LIN {X 0,Y 556.816,Z 344.275,A -85,B 0,C 180,E1 26754.409,E2 26754.409} C_VEL
LIN {X 0,Y 555.686,Z 542.378,A -85,B 0,C 180,E1 26751.669,E2 26751.669} C_VEL
LIN {X 0,Y 555.397,Z 561.24,A -85,B 0,C 180,E1 26751.213,E2 26751.213} C_VEL
LIN {X 0,Y 554.964,Z 579.491,A -85,B 0,C 180,E1 26750.568,E2 26750.568} C_VEL
LIN {X 0,Y 554.492,Z 596.687,A -85,B 0,C 180,E1 26749.755,E2 26749.755} C_VEL
LIN {X 0,Y 553.933,Z 616.269,A -85,B 0,C 180,E1 26748.582,E2 26748.582} C_VEL
LIN {X 0,Y 553.499,Z 632.409,A -85,B 0,C 180,E1 26747.395,E2 26747.395} C_VEL
LIN {X 0,Y 553.09,Z 647.422,A -85,B 0,C 180,E1 26746.056,E2 26746.056} C_VEL
LIN {X 0,Y 552.732,Z 661.164,A -85,B 0,C 180,E1 26744.582,E2 26744.582} C_VEL
LIN {X 0,Y 552.457,Z 672.902,A -85,B 0,C 180,E1 26743.075,E2 26743.075} C_VEL
LIN {X 0,Y 552.23,Z 683.866,A -85,B 0,C 180,E1 26741.382,E2 26741.382} C_VEL
LIN {X 0,Y 552.076,Z 693.318,A -85,B 0,C 180,E1 26739.591,E2 26739.591} C_VEL
LIN {X 0,Y 551.986,Z 700.982,A -85,B 0,C 180,E1 26737.765,E2 26737.765} C_VEL
LIN {X 0,Y 551.932,Z 707.192,A -85,B 0,C 180,E1 26735.822,E2 26735.822} C_VEL
LIN {X 0,Y 551.92,Z 711.605,A -85,B 0,C 180,E1 26733.843,E2 26733.843} C_VEL
LIN {X 0,Y 551.914,Z 714.178,A -85,B 0,C 180,E1 26731.869,E2 26731.869} C_VEL
LIN {X 0,Y 551.916,Z 714.992,A -85,B 0,C 180,E1 26729.896,E2 26729.896} C_VEL
LIN {X 0,Y 551.917,Z 714.065,A -85,B 0,C 180,E1 26727.924,E2 26727.924} C_VEL
LIN {X 0,Y 551.921,Z 711.376,A -85,B 0,C 180,E1 26725.949,E2 26725.949} C_VEL
LIN {X 0,Y 551.937,Z 706.971,A -85,B 0,C 180,E1 26724.011,E2 26724.011} C_VEL
LIN {X 0,Y 551.988,Z 700.76,A -85,B 0,C 180,E1 26722.088,E2 26722.088} C_VEL
LIN {X 0,Y 552.077,Z 693.245,A -85,B 0,C 180,E1 26720.304,E2 26720.304} C_VEL
LIN {X 0,Y 552.231,Z 683.772,A -85,B 0,C 180,E1 26718.512,E2 26718.512} C_VEL
LIN {X 0,Y 552.458,Z 672.783,A -85,B 0,C 180,E1 26716.819,E2 26716.819} C_VEL
LIN {X 0,Y 552.755,Z 660.265,A -85,B 0,C 180,E1 26715.224,E2 26715.224} C_VEL
LIN {X 0,Y 553.124,Z 646.131,A -85,B 0,C 180,E1 26713.729,E2 26713.729} C_VEL
LIN {X 0,Y 553.539,Z 630.846,A -85,B 0,C 180,E1 26712.389,E2 26712.389} C_VEL
LIN {X 0,Y 553.959,Z 615.253,A -85,B 0,C 180,E1 26711.26,E2 26711.26} C_VEL
LIN {X 0,Y 554.497,Z 596.601,A -85,B 0,C 180,E1 26710.151,E2 26710.151} C_VEL
LIN {X 0,Y 554.987,Z 579.027,A -85,B 0,C 180,E1 26709.323,E2 26709.323} C_VEL
LIN {X 0,Y 555.409,Z 560.565,A -85,B 0,C 180,E1 26708.677,E2 26708.677} C_VEL
LIN {X 0,Y 555.693,Z 541.746,A -85,B 0,C 180,E1 26708.23,E2 26708.23} C_VEL
LIN {X 0,Y 556.819,Z 343.095,A -85,B 0,C 180,E1 26705.485,E2 26705.485} C_VEL
LIN {X 0,Y 555.247,Z 334.788,A -85,B 0,C 180,E1 26705.25,E2 26705.25} C_VEL
LIN {X 0,Y 556.018,Z 305.385,A -85,B 0,C 180,E1 26702.475,E2 26702.475} C_VEL
LIN {X 0,Y 552.345,Z 293.887,A -85,B 0,C 180,E1 26701.069,E2 26701.069} C_VEL
LIN {X 0,Y 552.34,Z 293.681,A -85,B 0,C 180,E1 26697.846,E2 26697.846} C_VEL
LIN {X 0,Y 552.335,Z 293.677,A -85,B 0,C 180,E1 26694.474,E2 26694.474} C_VEL
LIN {X 0,Y 552.308,Z 293.678,A -85,B 0,C 180,E1 26691.119,E2 26691.119} C_VEL
LIN {X 0,Y 552.34,Z 293.682,A -85,B 0,C 180,E1 26687.811,E2 26687.811} C_VEL
LIN {X 0,Y 552.322,Z 293.677,A -85,B 0,C 180,E1 26684.474,E2 26684.474} C_VEL
LIN {X 0,Y 552.301,Z 293.684,A -85,B 0,C 180,E1 26681.084,E2 26681.084} C_VEL
LIN {X 0,Y 552.345,Z 293.682,A -85,B 0,C 180,E1 26677.855,E2 26677.855} C_VEL
LIN {X 0,Y 552.302,Z 293.681,A -85,B 0,C 180,E1 26674.545,E2 26674.545} C_VEL
LIN {X 0,Y 552.297,Z 293.685,A -85,B 0,C 180,E1 26671.099,E2 26671.099} C_VEL
LIN {X 0,Y 552.344,Z 293.681,A -85,B 0,C 180,E1 26667.842,E2 26667.842} C_VEL
LIN {X 0,Y 552.285,Z 293.679,A -85,B 0,C 180,E1 26664.607,E2 26664.607} C_VEL
LIN {X 0,Y 552.314,Z 293.685,A -85,B 0,C 180,E1 26661.338,E2 26661.338} C_VEL
LIN {X 0,Y 552.292,Z 293.682,A -85,B 0,C 180,E1 26658.252,E2 26658.252} C_VEL
LIN {X 0,Y 552.278,Z 293.681,A -85,B 0,C 180,E1 26654.897,E2 26654.897} C_VEL
LIN {X 0,Y 552.337,Z 293.685,A -85,B 0,C 180,E1 26651.676,E2 26651.676} C_VEL
LIN {X 0,Y 552.267,Z 293.68,A -85,B 0,C 180,E1 26648.433,E2 26648.433} C_VEL
LIN {X 0,Y 552.298,Z 293.687,A -85,B 0,C 180,E1 26645.194,E2 26645.194} C_VEL
LIN {X 0,Y 552.276,Z 293.682,A -85,B 0,C 180,E1 26642.075,E2 26642.075} C_VEL
LIN {X 0,Y 552.263,Z 293.686,A -85,B 0,C 180,E1 26638.755,E2 26638.755} C_VEL
LIN {X 0,Y 552.326,Z 293.685,A -85,B 0,C 180,E1 26635.536,E2 26635.536} C_VEL
LIN {X 0,Y 552.265,Z 293.683,A -85,B 0,C 180,E1 26632.406,E2 26632.406} C_VEL
LIN {X 0,Y 552.318,Z 293.686,A -85,B 0,C 180,E1 26629.148,E2 26629.148} C_VEL
LIN {X 0,Y 552.281,Z 293.681,A -85,B 0,C 180,E1 26626.014,E2 26626.014} C_VEL
LIN {X 0,Y 552.279,Z 293.683,A -85,B 0,C 180,E1 26622.566,E2 26622.566} C_VEL
LIN {X 0,Y 552.342,Z 293.686,A -85,B 0,C 180,E1 26619.33,E2 26619.33} C_VEL
LIN {X 0,Y 552.285,Z 293.683,A -85,B 0,C 180,E1 26616.096,E2 26616.096} C_VEL
LIN {X 0,Y 552.309,Z 293.68,A -85,B 0,C 180,E1 26612.741,E2 26612.741} C_VEL
LIN {X 0,Y 552.327,Z 293.686,A -85,B 0,C 180,E1 26609.504,E2 26609.504} C_VEL
LIN {X 0,Y 552.292,Z 293.684,A -85,B 0,C 180,E1 26606.195,E2 26606.195} C_VEL
LIN {X 0,Y 552.345,Z 293.677,A -85,B 0,C 180,E1 26602.93,E2 26602.93} C_VEL
LIN {X 0,Y 552.318,Z 293.684,A -85,B 0,C 180,E1 26599.603,E2 26599.603} C_VEL
LIN {X 0,Y 552.305,Z 293.684,A -85,B 0,C 180,E1 26596.245,E2 26596.245} C_VEL
LIN {X 0,Y 552.341,Z 293.676,A -85,B 0,C 180,E1 26593.002,E2 26593.002} C_VEL
LIN {X 0,Y 552.312,Z 293.674,A -85,B 0,C 180,E1 26589.702,E2 26589.702} C_VEL
LIN {X 0,Y 552.379,Z 293.923,A -85,B 0,C 180,E1 26586.704,E2 26586.704} C_VEL
LIN {X 0,Y 554.146,Z 298.811,A -85,B 0,C 180,E1 26586.242,E2 26586.242} C_VEL
LIN {X 0,Y 559.158,Z 310.667,A -85,B 0,C 180,E1 26585.196,E2 26585.196} C_VEL
LIN {X 0,Y 558.362,Z 353.988,A -85,B 0,C 180,E1 26582.614,E2 26582.614} C_VEL
LIN {X 0,Y 557.656,Z 390.963,A -85,B 0,C 180,E1 26580.436,E2 26580.436} C_VEL
LIN {X 0,Y 558.742,Z 400.337,A -85,B 0,C 180,E1 26580.232,E2 26580.232} C_VEL
LIN {X 0,Y 557.381,Z 635.152,A -85,B 0,C 180,E1 26576.937,E2 26576.937} C_VEL
LIN {X 0,Y 557.116,Z 659.61,A -85,B 0,C 180,E1 26576.529,E2 26576.529} C_VEL
LIN {X 0,Y 556.72,Z 680.633,A -85,B 0,C 180,E1 26575.975,E2 26575.975} C_VEL
LIN {X 0,Y 556.289,Z 700.028,A -85,B 0,C 180,E1 26575.274,E2 26575.274} C_VEL
LIN {X 0,Y 555.753,Z 719.239,A -85,B 0,C 180,E1 26574.386,E2 26574.386} C_VEL
LIN {X 0,Y 555.148,Z 738.316,A -85,B 0,C 180,E1 26573.286,E2 26573.286} C_VEL
LIN {X 0,Y 554.551,Z 756.388,A -85,B 0,C 180,E1 26572.025,E2 26572.025} C_VEL
LIN {X 0,Y 553.976,Z 773.443,A -85,B 0,C 180,E1 26570.606,E2 26570.606} C_VEL
LIN {X 0,Y 553.441,Z 789.448,A -85,B 0,C 180,E1 26569.031,E2 26569.031} C_VEL
LIN {X 0,Y 552.984,Z 804.238,A -85,B 0,C 180,E1 26567.315,E2 26567.315} C_VEL
LIN {X 0,Y 552.622,Z 817.278,A -85,B 0,C 180,E1 26565.531,E2 26565.531} C_VEL
LIN {X 0,Y 552.359,Z 828.534,A -85,B 0,C 180,E1 26563.717,E2 26563.717} C_VEL
LIN {X 0,Y 552.147,Z 838.91,A -85,B 0,C 180,E1 26561.701,E2 26561.701} C_VEL
LIN {X 0,Y 552.024,Z 847.28,A -85,B 0,C 180,E1 26559.697,E2 26559.697} C_VEL
LIN {X 0,Y 551.959,Z 854.202,A -85,B 0,C 180,E1 26557.599,E2 26557.599} C_VEL
LIN {X 0,Y 551.92,Z 859.556,A -85,B 0,C 180,E1 26555.405,E2 26555.405} C_VEL
LIN {X 0,Y 551.909,Z 862.942,A -85,B 0,C 180,E1 26553.323,E2 26553.323} C_VEL
LIN {X 0,Y 551.911,Z 864.759,A -85,B 0,C 180,E1 26551.142,E2 26551.142} C_VEL
LIN {X 0,Y 551.915,Z 864.783,A -85,B 0,C 180,E1 26548.962,E2 26548.962} C_VEL
LIN {X 0,Y 551.914,Z 863.169,A -85,B 0,C 180,E1 26546.885,E2 26546.885} C_VEL
LIN {X 0,Y 551.921,Z 859.76,A -85,B 0,C 180,E1 26544.699,E2 26544.699} C_VEL
LIN {X 0,Y 551.952,Z 854.809,A -85,B 0,C 180,E1 26542.611,E2 26542.611} C_VEL
LIN {X 0,Y 552.022,Z 848.49,A -85,B 0,C 180,E1 26540.618,E2 26540.618} C_VEL
LIN {X 0,Y 552.138,Z 839.875,A -85,B 0,C 180,E1 26538.51,E2 26538.51} C_VEL
LIN {X 0,Y 552.321,Z 830.266,A -85,B 0,C 180,E1 26536.602,E2 26536.602} C_VEL
LIN {X 0,Y 552.585,Z 818.607,A -85,B 0,C 180,E1 26534.67,E2 26534.67} C_VEL
LIN {X 0,Y 552.945,Z 805.602,A -85,B 0,C 180,E1 26532.858,E2 26532.858} C_VEL
LIN {X 0,Y 553.393,Z 790.965,A -85,B 0,C 180,E1 26531.131,E2 26531.131} C_VEL
LIN {X 0,Y 553.892,Z 775.855,A -85,B 0,C 180,E1 26529.611,E2 26529.611} C_VEL
LIN {X 0,Y 554.455,Z 759.284,A -85,B 0,C 180,E1 26528.193,E2 26528.193} C_VEL
LIN {X 0,Y 555.07,Z 740.902,A -85,B 0,C 180,E1 26526.879,E2 26526.879} C_VEL
LIN {X 0,Y 555.652,Z 722.284,A -85,B 0,C 180,E1 26525.779,E2 26525.779} C_VEL
LIN {X 0,Y 556.159,Z 704.004,A -85,B 0,C 180,E1 26524.896,E2 26524.896} C_VEL
LIN {X 0,Y 556.654,Z 683.569,A -85,B 0,C 180,E1 26524.118,E2 26524.118} C_VEL
LIN {X 0,Y 557.081,Z 663.506,A -85,B 0,C 180,E1 26523.556,E2 26523.556} C_VEL
LIN {X 0,Y 557.344,Z 642.37,A -85,B 0,C 180,E1 26523.163,E2 26523.163} C_VEL
LIN {X 0,Y 558.712,Z 404.697,A -85,B 0,C 180,E1 26519.829,E2 26519.829} C_VEL
LIN {X 0,Y 558.481,Z 396.637,A -85,B 0,C 180,E1 26519.698,E2 26519.698} C_VEL
LIN {X 0,Y 557.585,Z 389.593,A -85,B 0,C 180,E1 26519.505,E2 26519.505} C_VEL
LIN {X 0,Y 558.839,Z 332.018,A -85,B 0,C 180,E1 26516.068,E2 26516.068} C_VEL
LIN {X 0,Y 558.964,Z 309.864,A -85,B 0,C 180,E1 26514.743,E2 26514.743} C_VEL
LIN {X 0,Y 552.405,Z 294.092,A -85,B 0,C 180,E1 26513.324,E2 26513.324} C_VEL
LIN {X 0,Y 552.339,Z 293.671,A -85,B 0,C 180,E1 26512.969,E2 26512.969} C_VEL
LIN {X 0,Y 552.316,Z 293.676,A -85,B 0,C 180,E1 26509.653,E2 26509.653} C_VEL
LIN {X 0,Y 552.31,Z 293.676,A -85,B 0,C 180,E1 26506.246,E2 26506.246} C_VEL
LIN {X 0,Y 552.344,Z 293.682,A -85,B 0,C 180,E1 26503.004,E2 26503.004} C_VEL
LIN {X 0,Y 552.302,Z 293.683,A -85,B 0,C 180,E1 26499.702,E2 26499.702} C_VEL
LIN {X 0,Y 552.307,Z 293.672,A -85,B 0,C 180,E1 26496.297,E2 26496.297} C_VEL
LIN {X 0,Y 552.34,Z 293.682,A -85,B 0,C 180,E1 26493.016,E2 26493.016} C_VEL
LIN {X 0,Y 552.29,Z 293.685,A -85,B 0,C 180,E1 26489.739,E2 26489.739} C_VEL
LIN {X 0,Y 552.326,Z 293.687,A -85,B 0,C 180,E1 26486.444,E2 26486.444} C_VEL
LIN {X 0,Y 552.304,Z 293.681,A -85,B 0,C 180,E1 26483.244,E2 26483.244} C_VEL
LIN {X 0,Y 552.284,Z 293.685,A -85,B 0,C 180,E1 26479.898,E2 26479.898} C_VEL
LIN {X 0,Y 552.345,Z 293.684,A -85,B 0,C 180,E1 26476.619,E2 26476.619} C_VEL
LIN {X 0,Y 552.277,Z 293.679,A -85,B 0,C 180,E1 26473.399,E2 26473.399} C_VEL
LIN {X 0,Y 552.284,Z 293.685,A -85,B 0,C 180,E1 26469.992,E2 26469.992} C_VEL
LIN {X 0,Y 552.307,Z 293.682,A -85,B 0,C 180,E1 26466.862,E2 26466.862} C_VEL
LIN {X 0,Y 552.263,Z 293.684,A -85,B 0,C 180,E1 26463.633,E2 26463.633} C_VEL
LIN {X 0,Y 552.332,Z 293.688,A -85,B 0,C 180,E1 26460.415,E2 26460.415} C_VEL
LIN {X 0,Y 552.261,Z 293.683,A -85,B 0,C 180,E1 26457.198,E2 26457.198} C_VEL
LIN {X 0,Y 552.27,Z 293.687,A -85,B 0,C 180,E1 26453.764,E2 26453.764} C_VEL
LIN {X 0,Y 552.286,Z 293.681,A -85,B 0,C 180,E1 26450.833,E2 26450.833} C_VEL
LIN {X 0,Y 552.268,Z 293.686,A -85,B 0,C 180,E1 26447.558,E2 26447.558} C_VEL
LIN {X 0,Y 552.34,Z 293.683,A -85,B 0,C 180,E1 26444.352,E2 26444.352} C_VEL
LIN {X 0,Y 552.276,Z 293.684,A -85,B 0,C 180,E1 26441.091,E2 26441.091} C_VEL
LIN {X 0,Y 552.301,Z 293.685,A -85,B 0,C 180,E1 26437.767,E2 26437.767} C_VEL
LIN {X 0,Y 552.312,Z 293.681,A -85,B 0,C 180,E1 26434.593,E2 26434.593} C_VEL
LIN {X 0,Y 552.299,Z 293.687,A -85,B 0,C 180,E1 26432.738,E2 26432.738} C_VEL
LIN {X 0,Y 551.36,Z 293.809,A -85,B 0,C 180,E1 26431.938,E2 26431.938} C_VEL
LIN {X 0,Y 544.881,Z 294.609,A -85,B 0,C 180,E1 26429.694,E2 26429.694} C_VEL
LIN {X 0,Y 544.346,Z 294.673,A -85,B 0,C 180,E1 26429.109,E2 26429.109} C_VEL
LIN {X 0,Y 544.389,Z 294.67,A -85,B 0,C 180,E1 26425.804,E2 26425.804} C_VEL
LIN {X 0,Y 544.381,Z 294.675,A -85,B 0,C 180,E1 26422.507,E2 26422.507} C_VEL
LIN {X 0,Y 544.357,Z 294.672,A -85,B 0,C 180,E1 26419.164,E2 26419.164} C_VEL
LIN {X 0,Y 544.405,Z 294.667,A -85,B 0,C 180,E1 26415.887,E2 26415.887} C_VEL
LIN {X 0,Y 544.376,Z 294.665,A -85,B 0,C 180,E1 26412.523,E2 26412.523} C_VEL
LIN {X 0,Y 544.368,Z 294.665,A -85,B 0,C 180,E1 26409.184,E2 26409.184} C_VEL
LIN {X 0,Y 544.404,Z 294.669,A -85,B 0,C 180,E1 26405.864,E2 26405.864} C_VEL
LIN {X 0,Y 544.38,Z 294.676,A -85,B 0,C 180,E1 26402.537,E2 26402.537} C_VEL
LIN {X 0,Y 544.416,Z 294.861,A -85,B 0,C 180,E1 26399.297,E2 26399.297} C_VEL
LIN {X 0,Y 548.778,Z 308.855,A -85,B 0,C 180,E1 26397.566,E2 26397.566} C_VEL
LIN {X 0,Y 548.006,Z 335.919,A -85,B 0,C 180,E1 26395.02,E2 26395.02} C_VEL
LIN {X 0,Y 549.744,Z 345.387,A -85,B 0,C 180,E1 26394.785,E2 26394.785} C_VEL
LIN {X 0,Y 548.559,Z 542.987,A -85,B 0,C 180,E1 26392.041,E2 26392.041} C_VEL
LIN {X 0,Y 548.263,Z 561.882,A -85,B 0,C 180,E1 26391.584,E2 26391.584} C_VEL
LIN {X 0,Y 547.817,Z 579.557,A -85,B 0,C 180,E1 26390.96,E2 26390.96} C_VEL
LIN {X 0,Y 547.296,Z 596.827,A -85,B 0,C 180,E1 26390.146,E2 26390.146} C_VEL
LIN {X 0,Y 546.679,Z 613.249,A -85,B 0,C 180,E1 26389.165,E2 26389.165} C_VEL
LIN {X 0,Y 546.031,Z 629.329,A -85,B 0,C 180,E1 26387.971,E2 26387.971} C_VEL
LIN {X 0,Y 545.411,Z 644.251,A -85,B 0,C 180,E1 26386.617,E2 26386.617} C_VEL
LIN {X 0,Y 544.925,Z 659.491,A -85,B 0,C 180,E1 26384.993,E2 26384.993} C_VEL
LIN {X 0,Y 544.571,Z 672.136,A -85,B 0,C 180,E1 26383.376,E2 26383.376} C_VEL
LIN {X 0,Y 544.302,Z 683.234,A -85,B 0,C 180,E1 26381.657,E2 26381.657} C_VEL
LIN {X 0,Y 544.121,Z 692.806,A -85,B 0,C 180,E1 26379.84,E2 26379.84} C_VEL
LIN {X 0,Y 544.003,Z 700.413,A -85,B 0,C 180,E1 26378.029,E2 26378.029} C_VEL
LIN {X 0,Y 543.946,Z 706.59,A -85,B 0,C 180,E1 26376.12,E2 26376.12} C_VEL
LIN {X 0,Y 543.921,Z 710.996,A -85,B 0,C 180,E1 26374.217,E2 26374.217} C_VEL
LIN {X 0,Y 543.913,Z 713.744,A -85,B 0,C 180,E1 26372.318,E2 26372.318} C_VEL
LIN {X 0,Y 543.909,Z 714.928,A -85,B 0,C 180,E1 26370.316,E2 26370.316} C_VEL
LIN {X 0,Y 543.913,Z 714.376,A -85,B 0,C 180,E1 26368.315,E2 26368.315} C_VEL
LIN {X 0,Y 543.911,Z 712.229,A -85,B 0,C 180,E1 26366.417,E2 26366.417} C_VEL
LIN {X 0,Y 543.932,Z 708.459,A -85,B 0,C 180,E1 26364.515,E2 26364.515} C_VEL
LIN {X 0,Y 543.974,Z 702.972,A -85,B 0,C 180,E1 26362.608,E2 26362.608} C_VEL
LIN {X 0,Y 544.075,Z 695.621,A -85,B 0,C 180,E1 26360.694,E2 26360.694} C_VEL
LIN {X 0,Y 544.235,Z 686.506,A -85,B 0,C 180,E1 26358.831,E2 26358.831} C_VEL
LIN {X 0,Y 544.463,Z 676.445,A -85,B 0,C 180,E1 26357.162,E2 26357.162} C_VEL
LIN {X 0,Y 544.769,Z 664.701,A -85,B 0,C 180,E1 26355.546,E2 26355.546} C_VEL
LIN {X 0,Y 545.161,Z 651.496,A -85,B 0,C 180,E1 26354.032,E2 26354.032} C_VEL
LIN {X 0,Y 545.774,Z 635.715,A -85,B 0,C 180,E1 26352.484,E2 26352.484} C_VEL
LIN {X 0,Y 546.393,Z 620.716,A -85,B 0,C 180,E1 26351.268,E2 26351.268} C_VEL
LIN {X 0,Y 547.021,Z 604.25,A -85,B 0,C 180,E1 26350.181,E2 26350.181} C_VEL
LIN {X 0,Y 547.584,Z 587.755,A -85,B 0,C 180,E1 26349.31,E2 26349.31} C_VEL
LIN {X 0,Y 548.078,Z 569.85,A -85,B 0,C 180,E1 26348.584,E2 26348.584} C_VEL
LIN {X 0,Y 548.441,Z 551.518,A -85,B 0,C 180,E1 26348.051,E2 26348.051} C_VEL
LIN {X 0,Y 548.652,Z 532.068,A -85,B 0,C 180,E1 26347.695,E2 26347.695} C_VEL
LIN {X 0,Y 549.626,Z 343.643,A -85,B 0,C 180,E1 26345.094,E2 26345.094} C_VEL
LIN {X 0,Y 547.949,Z 335.49,A -85,B 0,C 180,E1 26344.869,E2 26344.869} C_VEL
LIN {X 0,Y 548.672,Z 308.058,A -85,B 0,C 180,E1 26342.257,E2 26342.257} C_VEL
LIN {X 0,Y 544.419,Z 294.84,A -85,B 0,C 180,E1 26340.606,E2 26340.606} C_VEL
LIN {X 0,Y 544.375,Z 294.675,A -85,B 0,C 180,E1 26337.193,E2 26337.193} C_VEL
LIN {X 0,Y 544.4,Z 294.672,A -85,B 0,C 180,E1 26333.876,E2 26333.876} C_VEL
LIN {X 0,Y 544.393,Z 294.662,A -85,B 0,C 180,E1 26330.48,E2 26330.48} C_VEL
LIN {X 0,Y 544.367,Z 294.663,A -85,B 0,C 180,E1 26327.127,E2 26327.127} C_VEL
LIN {X 0,Y 544.405,Z 294.671,A -85,B 0,C 180,E1 26323.8,E2 26323.8} C_VEL
LIN {X 0,Y 544.381,Z 294.669,A -85,B 0,C 180,E1 26320.418,E2 26320.418} C_VEL
LIN {X 0,Y 544.36,Z 294.674,A -85,B 0,C 180,E1 26317.046,E2 26317.046} C_VEL
LIN {X 0,Y 544.403,Z 294.67,A -85,B 0,C 180,E1 26313.699,E2 26313.699} C_VEL
LIN {X 0,Y 544.361,Z 294.671,A -85,B 0,C 180,E1 26310.461,E2 26310.461} C_VEL
LIN {X 0,Y 544.354,Z 294.675,A -85,B 0,C 180,E1 26307.025,E2 26307.025} C_VEL
LIN {X 0,Y 544.404,Z 294.668,A -85,B 0,C 180,E1 26303.717,E2 26303.717} C_VEL
LIN {X 0,Y 544.345,Z 294.671,A -85,B 0,C 180,E1 26300.488,E2 26300.488} C_VEL
LIN {X 0,Y 544.352,Z 294.676,A -85,B 0,C 180,E1 26297.091,E2 26297.091} C_VEL
LIN {X 0,Y 544.376,Z 294.667,A -85,B 0,C 180,E1 26293.923,E2 26293.923} C_VEL
LIN {X 0,Y 544.33,Z 294.675,A -85,B 0,C 180,E1 26290.676,E2 26290.676} C_VEL
LIN {X 0,Y 544.382,Z 294.675,A -85,B 0,C 180,E1 26287.387,E2 26287.387} C_VEL
LIN {X 0,Y 544.331,Z 294.675,A -85,B 0,C 180,E1 26284.214,E2 26284.214} C_VEL
LIN {X 0,Y 544.328,Z 294.677,A -85,B 0,C 180,E1 26280.842,E2 26280.842} C_VEL
LIN {X 0,Y 544.358,Z 294.674,A -85,B 0,C 180,E1 26277.79,E2 26277.79} C_VEL
LIN {X 0,Y 544.324,Z 294.676,A -85,B 0,C 180,E1 26274.519,E2 26274.519} C_VEL
LIN {X 0,Y 544.394,Z 294.67,A -85,B 0,C 180,E1 26271.338,E2 26271.338} C_VEL
LIN {X 0,Y 544.336,Z 294.676,A -85,B 0,C 180,E1 26268.128,E2 26268.128} C_VEL
LIN {X 0,Y 544.343,Z 294.675,A -85,B 0,C 180,E1 26264.644,E2 26264.644} C_VEL
LIN {X 0,Y 544.4,Z 294.669,A -85,B 0,C 180,E1 26261.382,E2 26261.382} C_VEL
LIN {X 0,Y 544.344,Z 294.675,A -85,B 0,C 180,E1 26258.107,E2 26258.107} C_VEL
LIN {X 0,Y 544.37,Z 294.673,A -85,B 0,C 180,E1 26254.779,E2 26254.779} C_VEL
LIN {X 0,Y 544.38,Z 294.673,A -85,B 0,C 180,E1 26251.595,E2 26251.595} C_VEL
LIN {X 0,Y 544.353,Z 294.672,A -85,B 0,C 180,E1 26248.256,E2 26248.256} C_VEL
LIN {X 0,Y 544.399,Z 294.657,A -85,B 0,C 180,E1 26244.91,E2 26244.91} C_VEL
LIN {X 0,Y 544.377,Z 294.673,A -85,B 0,C 180,E1 26241.625,E2 26241.625} C_VEL
LIN {X 0,Y 544.361,Z 294.657,A -85,B 0,C 180,E1 26238.219,E2 26238.219} C_VEL
LIN {X 0,Y 544.405,Z 294.666,A -85,B 0,C 180,E1 26234.997,E2 26234.997} C_VEL
LIN {X 0,Y 544.379,Z 294.677,A -85,B 0,C 180,E1 26231.623,E2 26231.623} C_VEL
LIN {X 0,Y 544.374,Z 294.678,A -85,B 0,C 180,E1 26228.177,E2 26228.177} C_VEL
LIN {X 0,Y 544.442,Z 294.964,A -85,B 0,C 180,E1 26227.17,E2 26227.17} C_VEL
LIN {X 0,Y 548.919,Z 306.372,A -85,B 0,C 180,E1 26226.115,E2 26226.115} C_VEL
LIN {X 0,Y 552.058,Z 313.827,A -85,B 0,C 180,E1 26225.452,E2 26225.452} C_VEL
LIN {X 0,Y 551.041,Z 367.835,A -85,B 0,C 180,E1 26222.238,E2 26222.238} C_VEL
LIN {X 0,Y 550.595,Z 391.148,A -85,B 0,C 180,E1 26220.865,E2 26220.865} C_VEL
LIN {X 0,Y 551.824,Z 401.323,A -85,B 0,C 180,E1 26220.637,E2 26220.637} C_VEL
LIN {X 0,Y 550.243,Z 636.347,A -85,B 0,C 180,E1 26217.298,E2 26217.298} C_VEL
LIN {X 0,Y 549.945,Z 659.772,A -85,B 0,C 180,E1 26216.898,E2 26216.898} C_VEL
LIN {X 0,Y 549.493,Z 680.847,A -85,B 0,C 180,E1 26216.336,E2 26216.336} C_VEL
LIN {X 0,Y 548.978,Z 700.613,A -85,B 0,C 180,E1 26215.609,E2 26215.609} C_VEL
LIN {X 0,Y 548.378,Z 719.24,A -85,B 0,C 180,E1 26214.736,E2 26214.736} C_VEL
LIN {X 0,Y 547.692,Z 738.326,A -85,B 0,C 180,E1 26213.622,E2 26213.622} C_VEL
LIN {X 0,Y 546.999,Z 756.39,A -85,B 0,C 180,E1 26212.346,E2 26212.346} C_VEL
LIN {X 0,Y 546.323,Z 773.443,A -85,B 0,C 180,E1 26210.908,E2 26210.908} C_VEL
LIN {X 0,Y 545.715,Z 789.202,A -85,B 0,C 180,E1 26209.338,E2 26209.338} C_VEL
LIN {X 0,Y 545.179,Z 803.91,A -85,B 0,C 180,E1 26207.614,E2 26207.614} C_VEL
LIN {X 0,Y 544.775,Z 816.573,A -85,B 0,C 180,E1 26205.87,E2 26205.87} C_VEL
LIN {X 0,Y 544.438,Z 828.535,A -85,B 0,C 180,E1 26203.92,E2 26203.92} C_VEL
LIN {X 0,Y 544.188,Z 838.909,A -85,B 0,C 180,E1 26201.875,E2 26201.875} C_VEL
LIN {X 0,Y 544.043,Z 847.279,A -85,B 0,C 180,E1 26199.841,E2 26199.841} C_VEL
LIN {X 0,Y 543.968,Z 854.202,A -85,B 0,C 180,E1 26197.711,E2 26197.711} C_VEL
LIN {X 0,Y 543.923,Z 859.556,A -85,B 0,C 180,E1 26195.485,E2 26195.485} C_VEL
LIN {X 0,Y 543.909,Z 862.942,A -85,B 0,C 180,E1 26193.372,E2 26193.372} C_VEL
LIN {X 0,Y 543.91,Z 864.759,A -85,B 0,C 180,E1 26191.159,E2 26191.159} C_VEL
LIN {X 0,Y 543.914,Z 864.783,A -85,B 0,C 180,E1 26188.947,E2 26188.947} C_VEL
LIN {X 0,Y 543.913,Z 863.168,A -85,B 0,C 180,E1 26186.839,E2 26186.839} C_VEL
LIN {X 0,Y 543.922,Z 859.761,A -85,B 0,C 180,E1 26184.621,E2 26184.621} C_VEL
LIN {X 0,Y 543.96,Z 854.81,A -85,B 0,C 180,E1 26182.501,E2 26182.501} C_VEL
LIN {X 0,Y 544.038,Z 848.49,A -85,B 0,C 180,E1 26180.479,E2 26180.479} C_VEL
LIN {X 0,Y 544.175,Z 839.876,A -85,B 0,C 180,E1 26178.34,E2 26178.34} C_VEL
LIN {X 0,Y 544.394,Z 830.268,A -85,B 0,C 180,E1 26176.403,E2 26176.403} C_VEL
LIN {X 0,Y 544.705,Z 818.691,A -85,B 0,C 180,E1 26174.455,E2 26174.455} C_VEL
LIN {X 0,Y 545.128,Z 805.601,A -85,B 0,C 180,E1 26172.605,E2 26172.605} C_VEL
LIN {X 0,Y 545.651,Z 790.965,A -85,B 0,C 180,E1 26170.853,E2 26170.853} C_VEL
LIN {X 0,Y 546.252,Z 775.515,A -85,B 0,C 180,E1 26169.282,E2 26169.282} C_VEL
LIN {X 0,Y 546.907,Z 758.842,A -85,B 0,C 180,E1 26167.841,E2 26167.841} C_VEL
LIN {X 0,Y 547.591,Z 740.898,A -85,B 0,C 180,E1 26166.544,E2 26166.544} C_VEL
LIN {X 0,Y 548.224,Z 723.385,A -85,B 0,C 180,E1 26165.492,E2 26165.492} C_VEL
LIN {X 0,Y 548.857,Z 704.001,A -85,B 0,C 180,E1 26164.538,E2 26164.538} C_VEL
LIN {X 0,Y 549.412,Z 683.823,A -85,B 0,C 180,E1 26163.76,E2 26163.76} C_VEL
LIN {X 0,Y 549.903,Z 663.669,A -85,B 0,C 180,E1 26163.187,E2 26163.187} C_VEL
LIN {X 0,Y 550.205,Z 642.495,A -85,B 0,C 180,E1 26162.788,E2 26162.788} C_VEL
LIN {X 0,Y 551.793,Z 405.141,A -85,B 0,C 180,E1 26159.417,E2 26159.417} C_VEL
LIN {X 0,Y 551.569,Z 397.823,A -85,B 0,C 180,E1 26159.295,E2 26159.295} C_VEL
LIN {X 0,Y 550.502,Z 389.593,A -85,B 0,C 180,E1 26159.07,E2 26159.07} C_VEL
LIN {X 0,Y 551.484,Z 344.188,A -85,B 0,C 180,E1 26156.367,E2 26156.367} C_VEL
LIN {X 0,Y 551.986,Z 313.279,A -85,B 0,C 180,E1 26154.51,E2 26154.51} C_VEL
LIN {X 0,Y 544.464,Z 295.085,A -85,B 0,C 180,E1 26152.844,E2 26152.844} C_VEL
LIN {X 0,Y 544.387,Z 294.664,A -85,B 0,C 180,E1 26152.508,E2 26152.508} C_VEL
LIN {X 0,Y 544.405,Z 294.663,A -85,B 0,C 180,E1 26149.17,E2 26149.17} C_VEL
LIN {X 0,Y 544.365,Z 294.666,A -85,B 0,C 180,E1 26145.885,E2 26145.885} C_VEL
LIN {X 0,Y 544.388,Z 294.66,A -85,B 0,C 180,E1 26142.523,E2 26142.523} C_VEL
LIN {X 0,Y 544.401,Z 294.67,A -85,B 0,C 180,E1 26139.183,E2 26139.183} C_VEL
LIN {X 0,Y 544.354,Z 294.66,A -85,B 0,C 180,E1 26135.869,E2 26135.869} C_VEL
LIN {X 0,Y 544.393,Z 294.676,A -85,B 0,C 180,E1 26132.542,E2 26132.542} C_VEL
LIN {X 0,Y 544.376,Z 294.672,A -85,B 0,C 180,E1 26129.246,E2 26129.246} C_VEL
LIN {X 0,Y 544.349,Z 294.675,A -85,B 0,C 180,E1 26125.922,E2 26125.922} C_VEL
LIN {X 0,Y 544.409,Z 294.668,A -85,B 0,C 180,E1 26122.686,E2 26122.686} C_VEL
LIN {X 0,Y 544.348,Z 294.672,A -85,B 0,C 180,E1 26119.418,E2 26119.418} C_VEL
LIN {X 0,Y 544.349,Z 294.676,A -85,B 0,C 180,E1 26115.993,E2 26115.993} C_VEL
LIN {X 0,Y 544.397,Z 294.666,A -85,B 0,C 180,E1 26112.732,E2 26112.732} C_VEL
LIN {X 0,Y 544.333,Z 294.673,A -85,B 0,C 180,E1 26109.474,E2 26109.474} C_VEL
LIN {X 0,Y 544.366,Z 294.677,A -85,B 0,C 180,E1 26106.221,E2 26106.221} C_VEL
LIN {X 0,Y 544.342,Z 294.672,A -85,B 0,C 180,E1 26103.053,E2 26103.053} C_VEL
LIN {X 0,Y 544.324,Z 294.677,A -85,B 0,C 180,E1 26099.684,E2 26099.684} C_VEL
LIN {X 0,Y 544.383,Z 294.669,A -85,B 0,C 180,E1 26096.525,E2 26096.525} C_VEL
LIN {X 0,Y 544.321,Z 294.676,A -85,B 0,C 180,E1 26093.354,E2 26093.354} C_VEL
LIN {X 0,Y 544.376,Z 294.675,A -85,B 0,C 180,E1 26090.165,E2 26090.165} C_VEL
LIN {X 0,Y 544.335,Z 294.675,A -85,B 0,C 180,E1 26087.05,E2 26087.05} C_VEL
LIN {X 0,Y 544.338,Z 294.675,A -85,B 0,C 180,E1 26083.568,E2 26083.568} C_VEL
LIN {X 0,Y 544.397,Z 294.669,A -85,B 0,C 180,E1 26080.36,E2 26080.36} C_VEL
LIN {X 0,Y 544.34,Z 294.675,A -85,B 0,C 180,E1 26077.082,E2 26077.082} C_VEL
LIN {X 0,Y 544.361,Z 294.673,A -85,B 0,C 180,E1 26073.677,E2 26073.677} C_VEL
LIN {X 0,Y 544.38,Z 294.672,A -85,B 0,C 180,E1 26070.512,E2 26070.512} C_VEL
LIN {X 0,Y 544.346,Z 294.673,A -85,B 0,C 180,E1 26069.109,E2 26069.109} C_VEL
LIN {X 0,Y 543.375,Z 294.804,A -85,B 0,C 180,E1 26068.298,E2 26068.298} C_VEL
LIN {X 0,Y 536.878,Z 295.607,A -85,B 0,C 180,E1 26065.962,E2 26065.962} C_VEL
LIN {X 0,Y 536.42,Z 295.66,A -85,B 0,C 180,E1 26065.427,E2 26065.427} C_VEL
LIN {X 0,Y 536.466,Z 295.659,A -85,B 0,C 180,E1 26062.179,E2 26062.179} C_VEL
LIN {X 0,Y 536.421,Z 295.663,A -85,B 0,C 180,E1 26058.852,E2 26058.852} C_VEL
LIN {X 0,Y 536.433,Z 295.656,A -85,B 0,C 180,E1 26055.397,E2 26055.397} C_VEL
LIN {X 0,Y 536.464,Z 295.657,A -85,B 0,C 180,E1 26052.116,E2 26052.116} C_VEL
LIN {X 0,Y 536.426,Z 295.652,A -85,B 0,C 180,E1 26048.775,E2 26048.775} C_VEL
LIN {X 0,Y 536.442,Z 295.657,A -85,B 0,C 180,E1 26045.295,E2 26045.295} C_VEL
LIN {X 0,Y 536.463,Z 295.656,A -85,B 0,C 180,E1 26041.958,E2 26041.958} C_VEL
LIN {X 0,Y 536.499,Z 295.915,A -85,B 0,C 180,E1 26039.745,E2 26039.745} C_VEL
LIN {X 0,Y 541.485,Z 311.262,A -85,B 0,C 180,E1 26037.812,E2 26037.812} C_VEL
LIN {X 0,Y 540.72,Z 336.313,A -85,B 0,C 180,E1 26035.435,E2 26035.435} C_VEL
LIN {X 0,Y 542.697,Z 346.672,A -85,B 0,C 180,E1 26035.169,E2 26035.169} C_VEL
LIN {X 0,Y 541.466,Z 544.211,A -85,B 0,C 180,E1 26032.415,E2 26032.415} C_VEL
LIN {X 0,Y 541.155,Z 563.162,A -85,B 0,C 180,E1 26031.949,E2 26031.949} C_VEL
LIN {X 0,Y 540.667,Z 580.996,A -85,B 0,C 180,E1 26031.308,E2 26031.308} C_VEL
LIN {X 0,Y 540.083,Z 598.216,A -85,B 0,C 180,E1 26030.48,E2 26030.48} C_VEL
LIN {X 0,Y 539.356,Z 615.276,A -85,B 0,C 180,E1 26029.436,E2 26029.436} C_VEL
LIN {X 0,Y 538.667,Z 630.549,A -85,B 0,C 180,E1 26028.281,E2 26028.281} C_VEL
LIN {X 0,Y 537.958,Z 645.447,A -85,B 0,C 180,E1 26026.91,E2 26026.91} C_VEL
LIN {X 0,Y 537.315,Z 658.759,A -85,B 0,C 180,E1 26025.432,E2 26025.432} C_VEL
LIN {X 0,Y 536.769,Z 671.005,A -85,B 0,C 180,E1 26023.794,E2 26023.794} C_VEL
LIN {X 0,Y 536.337,Z 684.507,A -85,B 0,C 180,E1 26021.615,E2 26021.615} C_VEL
LIN {X 0,Y 536.133,Z 693.838,A -85,B 0,C 180,E1 26019.771,E2 26019.771} C_VEL
LIN {X 0,Y 536.006,Z 701.614,A -85,B 0,C 180,E1 26017.826,E2 26017.826} C_VEL
LIN {X 0,Y 535.94,Z 707.481,A -85,B 0,C 180,E1 26015.889,E2 26015.889} C_VEL
LIN {X 0,Y 535.92,Z 711.772,A -85,B 0,C 180,E1 26013.851,E2 26013.851} C_VEL
LIN {X 0,Y 535.913,Z 714.248,A -85,B 0,C 180,E1 26011.818,E2 26011.818} C_VEL
LIN {X 0,Y 535.913,Z 714.969,A -85,B 0,C 180,E1 26009.786,E2 26009.786} C_VEL
LIN {X 0,Y 535.916,Z 713.954,A -85,B 0,C 180,E1 26007.755,E2 26007.755} C_VEL
LIN {X 0,Y 535.922,Z 711.375,A -85,B 0,C 180,E1 26005.828,E2 26005.828} C_VEL
LIN {X 0,Y 535.947,Z 707.148,A -85,B 0,C 180,E1 26003.896,E2 26003.896} C_VEL
LIN {X 0,Y 536.013,Z 701.161,A -85,B 0,C 180,E1 26001.958,E2 26001.958} C_VEL
LIN {X 0,Y 536.136,Z 693.754,A -85,B 0,C 180,E1 26000.121,E2 26000.121} C_VEL
LIN {X 0,Y 536.341,Z 684.398,A -85,B 0,C 180,E1 25998.276,E2 25998.276} C_VEL
LIN {X 0,Y 536.794,Z 670.46,A -85,B 0,C 180,E1 25996.035,E2 25996.035} C_VEL
LIN {X 0,Y 537.325,Z 658.594,A -85,B 0,C 180,E1 25994.458,E2 25994.458} C_VEL
LIN {X 0,Y 537.971,Z 645.245,A -85,B 0,C 180,E1 25992.979,E2 25992.979} C_VEL
LIN {X 0,Y 538.681,Z 630.3,A -85,B 0,C 180,E1 25991.607,E2 25991.607} C_VEL
LIN {X 0,Y 539.414,Z 614.175,A -85,B 0,C 180,E1 25990.398,E2 25990.398} C_VEL
LIN {X 0,Y 540.101,Z 597.813,A -85,B 0,C 180,E1 25989.407,E2 25989.407} C_VEL
LIN {X 0,Y 540.692,Z 580.44,A -85,B 0,C 180,E1 25988.579,E2 25988.579} C_VEL
LIN {X 0,Y 541.172,Z 562.076,A -85,B 0,C 180,E1 25987.93,E2 25987.93} C_VEL
LIN {X 0,Y 541.473,Z 543.525,A -85,B 0,C 180,E1 25987.484,E2 25987.484} C_VEL
LIN {X 0,Y 542.586,Z 364.02,A -85,B 0,C 180,E1 25984.978,E2 25984.978} C_VEL
LIN {X 0,Y 542.483,Z 344.395,A -85,B 0,C 180,E1 25984.696,E2 25984.696} C_VEL
LIN {X 0,Y 540.658,Z 335.774,A -85,B 0,C 180,E1 25984.445,E2 25984.445} C_VEL
LIN {X 0,Y 541.472,Z 311.202,A -85,B 0,C 180,E1 25982.09,E2 25982.09} C_VEL
LIN {X 0,Y 536.494,Z 295.899,A -85,B 0,C 180,E1 25980.159,E2 25980.159} C_VEL
LIN {X 0,Y 536.439,Z 295.662,A -85,B 0,C 180,E1 25976.9,E2 25976.9} C_VEL
LIN {X 0,Y 536.442,Z 295.663,A -85,B 0,C 180,E1 25973.386,E2 25973.386} C_VEL
LIN {X 0,Y 536.462,Z 295.654,A -85,B 0,C 180,E1 25969.985,E2 25969.985} C_VEL
LIN {X 0,Y 536.436,Z 295.648,A -85,B 0,C 180,E1 25966.629,E2 25966.629} C_VEL
LIN {X 0,Y 536.428,Z 295.664,A -85,B 0,C 180,E1 25963.162,E2 25963.162} C_VEL
LIN {X 0,Y 536.467,Z 295.661,A -85,B 0,C 180,E1 25959.838,E2 25959.838} C_VEL
LIN {X 0,Y 536.431,Z 295.66,A -85,B 0,C 180,E1 25956.484,E2 25956.484} C_VEL
LIN {X 0,Y 536.42,Z 295.663,A -85,B 0,C 180,E1 25953.103,E2 25953.103} C_VEL
LIN {X 0,Y 536.469,Z 295.658,A -85,B 0,C 180,E1 25949.844,E2 25949.844} C_VEL
LIN {X 0,Y 536.413,Z 295.662,A -85,B 0,C 180,E1 25946.533,E2 25946.533} C_VEL
LIN {X 0,Y 536.414,Z 295.664,A -85,B 0,C 180,E1 25943.044,E2 25943.044} C_VEL
LIN {X 0,Y 536.466,Z 295.656,A -85,B 0,C 180,E1 25939.749,E2 25939.749} C_VEL
LIN {X 0,Y 536.401,Z 295.663,A -85,B 0,C 180,E1 25936.459,E2 25936.459} C_VEL
LIN {X 0,Y 536.407,Z 295.664,A -85,B 0,C 180,E1 25933.035,E2 25933.035} C_VEL
LIN {X 0,Y 536.433,Z 295.663,A -85,B 0,C 180,E1 25929.874,E2 25929.874} C_VEL
LIN {X 0,Y 536.387,Z 295.665,A -85,B 0,C 180,E1 25926.637,E2 25926.637} C_VEL
LIN {X 0,Y 536.443,Z 295.657,A -85,B 0,C 180,E1 25923.42,E2 25923.42} C_VEL
LIN {X 0,Y 536.385,Z 295.666,A -85,B 0,C 180,E1 25920.214,E2 25920.214} C_VEL
LIN {X 0,Y 536.39,Z 295.661,A -85,B 0,C 180,E1 25916.794,E2 25916.794} C_VEL
LIN {X 0,Y 536.446,Z 295.665,A -85,B 0,C 180,E1 25913.579,E2 25913.579} C_VEL
LIN {X 0,Y 536.39,Z 295.663,A -85,B 0,C 180,E1 25910.342,E2 25910.342} C_VEL
LIN {X 0,Y 536.435,Z 295.655,A -85,B 0,C 180,E1 25907.076,E2 25907.076} C_VEL
LIN {X 0,Y 536.414,Z 295.665,A -85,B 0,C 180,E1 25903.875,E2 25903.875} C_VEL
LIN {X 0,Y 536.405,Z 295.662,A -85,B 0,C 180,E1 25900.509,E2 25900.509} C_VEL
LIN {X 0,Y 536.467,Z 295.656,A -85,B 0,C 180,E1 25897.191,E2 25897.191} C_VEL
LIN {X 0,Y 536.417,Z 295.664,A -85,B 0,C 180,E1 25893.903,E2 25893.903} C_VEL
LIN {X 0,Y 536.42,Z 295.662,A -85,B 0,C 180,E1 25890.509,E2 25890.509} C_VEL
LIN {X 0,Y 536.468,Z 295.662,A -85,B 0,C 180,E1 25887.197,E2 25887.197} C_VEL
LIN {X 0,Y 536.419,Z 295.646,A -85,B 0,C 180,E1 25883.914,E2 25883.914} C_VEL
LIN {X 0,Y 536.434,Z 295.66,A -85,B 0,C 180,E1 25880.501,E2 25880.501} C_VEL
LIN {X 0,Y 536.463,Z 295.652,A -85,B 0,C 180,E1 25877.134,E2 25877.134} C_VEL
LIN {X 0,Y 536.432,Z 295.65,A -85,B 0,C 180,E1 25873.748,E2 25873.748} C_VEL
LIN {X 0,Y 536.436,Z 295.65,A -85,B 0,C 180,E1 25870.297,E2 25870.297} C_VEL
LIN {X 0,Y 536.468,Z 295.89,A -85,B 0,C 180,E1 25867.684,E2 25867.684} C_VEL
LIN {X 0,Y 537.386,Z 298.529,A -85,B 0,C 180,E1 25867.395,E2 25867.395} C_VEL
LIN {X 0,Y 544.954,Z 316.732,A -85,B 0,C 180,E1 25865.725,E2 25865.725} C_VEL
LIN {X 0,Y 543.784,Z 370.83,A -85,B 0,C 180,E1 25862.472,E2 25862.472} C_VEL
LIN {X 0,Y 543.515,Z 391.139,A -85,B 0,C 180,E1 25861.306,E2 25861.306} C_VEL
LIN {X 0,Y 544.931,Z 402.537,A -85,B 0,C 180,E1 25861.049,E2 25861.049} C_VEL
LIN {X 0,Y 543.124,Z 637.969,A -85,B 0,C 180,E1 25857.663,E2 25857.663} C_VEL
LIN {X 0,Y 542.789,Z 660.42,A -85,B 0,C 180,E1 25857.267,E2 25857.267} C_VEL
LIN {X 0,Y 542.279,Z 681.388,A -85,B 0,C 180,E1 25856.695,E2 25856.695} C_VEL
LIN {X 0,Y 541.676,Z 701.436,A -85,B 0,C 180,E1 25855.942,E2 25855.942} C_VEL
LIN {X 0,Y 540.985,Z 720.276,A -85,B 0,C 180,E1 25855.039,E2 25855.039} C_VEL
LIN {X 0,Y 540.22,Z 739.219,A -85,B 0,C 180,E1 25853.911,E2 25853.911} C_VEL
LIN {X 0,Y 539.435,Z 757.064,A -85,B 0,C 180,E1 25852.623,E2 25852.623} C_VEL
LIN {X 0,Y 538.666,Z 774.049,A -85,B 0,C 180,E1 25851.163,E2 25851.163} C_VEL
LIN {X 0,Y 537.963,Z 789.953,A -85,B 0,C 180,E1 25849.544,E2 25849.544} C_VEL
LIN {X 0,Y 537.346,Z 804.756,A -85,B 0,C 180,E1 25847.767,E2 25847.767} C_VEL
LIN {X 0,Y 536.86,Z 817.987,A -85,B 0,C 180,E1 25845.889,E2 25845.889} C_VEL
LIN {X 0,Y 536.505,Z 829.114,A -85,B 0,C 180,E1 25844.02,E2 25844.02} C_VEL
LIN {X 0,Y 536.225,Z 839.412,A -85,B 0,C 180,E1 25841.945,E2 25841.945} C_VEL
LIN {X 0,Y 536.056,Z 848.088,A -85,B 0,C 180,E1 25839.772,E2 25839.772} C_VEL
LIN {X 0,Y 535.974,Z 854.505,A -85,B 0,C 180,E1 25837.719,E2 25837.719} C_VEL
LIN {X 0,Y 535.928,Z 859.555,A -85,B 0,C 180,E1 25835.567,E2 25835.567} C_VEL
LIN {X 0,Y 535.91,Z 862.941,A -85,B 0,C 180,E1 25833.423,E2 25833.423} C_VEL
LIN {X 0,Y 535.909,Z 864.759,A -85,B 0,C 180,E1 25831.176,E2 25831.176} C_VEL
LIN {X 0,Y 535.915,Z 864.805,A -85,B 0,C 180,E1 25829.038,E2 25829.038} C_VEL
LIN {X 0,Y 535.914,Z 863.281,A -85,B 0,C 180,E1 25826.899,E2 25826.899} C_VEL
LIN {X 0,Y 535.924,Z 859.966,A -85,B 0,C 180,E1 25824.648,E2 25824.648} C_VEL
LIN {X 0,Y 535.965,Z 855.113,A -85,B 0,C 180,E1 25822.497,E2 25822.497} C_VEL
LIN {X 0,Y 536.055,Z 848.49,A -85,B 0,C 180,E1 25820.336,E2 25820.336} C_VEL
LIN {X 0,Y 536.214,Z 839.877,A -85,B 0,C 180,E1 25818.164,E2 25818.164} C_VEL
LIN {X 0,Y 536.475,Z 830.125,A -85,B 0,C 180,E1 25816.171,E2 25816.171} C_VEL
LIN {X 0,Y 536.835,Z 818.69,A -85,B 0,C 180,E1 25814.222,E2 25814.222} C_VEL
LIN {X 0,Y 537.324,Z 805.371,A -85,B 0,C 180,E1 25812.313,E2 25812.313} C_VEL
LIN {X 0,Y 537.923,Z 790.965,A -85,B 0,C 180,E1 25810.567,E2 25810.567} C_VEL
LIN {X 0,Y 538.596,Z 775.859,A -85,B 0,C 180,E1 25809.006,E2 25809.006} C_VEL
LIN {X 0,Y 539.375,Z 758.573,A -85,B 0,C 180,E1 25807.494,E2 25807.494} C_VEL
LIN {X 0,Y 540.137,Z 740.895,A -85,B 0,C 180,E1 25806.201,E2 25806.201} C_VEL
LIN {X 0,Y 540.87,Z 722.982,A -85,B 0,C 180,E1 25805.114,E2 25805.114} C_VEL
LIN {X 0,Y 541.577,Z 703.998,A -85,B 0,C 180,E1 25804.171,E2 25804.171} C_VEL
LIN {X 0,Y 542.2,Z 683.938,A -85,B 0,C 180,E1 25803.387,E2 25803.387} C_VEL
LIN {X 0,Y 542.749,Z 663.832,A -85,B 0,C 180,E1 25802.808,E2 25802.808} C_VEL
LIN {X 0,Y 543.092,Z 642.495,A -85,B 0,C 180,E1 25802.402,E2 25802.402} C_VEL
LIN {X 0,Y 544.906,Z 405.395,A -85,B 0,C 180,E1 25798.992,E2 25798.992} C_VEL
LIN {X 0,Y 544.666,Z 398.89,A -85,B 0,C 180,E1 25798.879,E2 25798.879} C_VEL
LIN {X 0,Y 543.416,Z 389.969,A -85,B 0,C 180,E1 25798.652,E2 25798.652} C_VEL
LIN {X 0,Y 544.565,Z 334.264,A -85,B 0,C 180,E1 25795.341,E2 25795.341} C_VEL
LIN {X 0,Y 544.752,Z 316.051,A -85,B 0,C 180,E1 25794.219,E2 25794.219} C_VEL
LIN {X 0,Y 536.504,Z 296.088,A -85,B 0,C 180,E1 25792.353,E2 25792.353} C_VEL
LIN {X 0,Y 536.431,Z 295.662,A -85,B 0,C 180,E1 25792.039,E2 25792.039} C_VEL
LIN {X 0,Y 536.464,Z 295.66,A -85,B 0,C 180,E1 25788.686,E2 25788.686} C_VEL
LIN {X 0,Y 536.462,Z 295.652,A -85,B 0,C 180,E1 25785.211,E2 25785.211} C_VEL
LIN {X 0,Y 536.422,Z 295.643,A -85,B 0,C 180,E1 25781.858,E2 25781.858} C_VEL
LIN {X 0,Y 536.448,Z 295.662,A -85,B 0,C 180,E1 25778.483,E2 25778.483} C_VEL
LIN {X 0,Y 536.458,Z 295.644,A -85,B 0,C 180,E1 25775.096,E2 25775.096} C_VEL
LIN {X 0,Y 536.415,Z 295.661,A -85,B 0,C 180,E1 25771.795,E2 25771.795} C_VEL
LIN {X 0,Y 536.455,Z 295.662,A -85,B 0,C 180,E1 25768.499,E2 25768.499} C_VEL
LIN {X 0,Y 536.439,Z 295.662,A -85,B 0,C 180,E1 25765.148,E2 25765.148} C_VEL
LIN {X 0,Y 536.407,Z 295.664,A -85,B 0,C 180,E1 25761.838,E2 25761.838} C_VEL
LIN {X 0,Y 536.461,Z 295.657,A -85,B 0,C 180,E1 25758.585,E2 25758.585} C_VEL
LIN {X 0,Y 536.406,Z 295.663,A -85,B 0,C 180,E1 25755.348,E2 25755.348} C_VEL
LIN {X 0,Y 536.4,Z 295.665,A -85,B 0,C 180,E1 25751.88,E2 25751.88} C_VEL
LIN {X 0,Y 536.459,Z 295.657,A -85,B 0,C 180,E1 25748.575,E2 25748.575} C_VEL
LIN {X 0,Y 536.391,Z 295.665,A -85,B 0,C 180,E1 25745.348,E2 25745.348} C_VEL
LIN {X 0,Y 536.4,Z 295.663,A -85,B 0,C 180,E1 25741.923,E2 25741.923} C_VEL
LIN {X 0,Y 536.415,Z 295.666,A -85,B 0,C 180,E1 25738.825,E2 25738.825} C_VEL
LIN {X 0,Y 536.38,Z 295.665,A -85,B 0,C 180,E1 25735.509,E2 25735.509} C_VEL
LIN {X 0,Y 536.449,Z 295.656,A -85,B 0,C 180,E1 25732.288,E2 25732.288} C_VEL
LIN {X 0,Y 536.396,Z 295.665,A -85,B 0,C 180,E1 25729.039,E2 25729.039} C_VEL
LIN {X 0,Y 536.399,Z 295.657,A -85,B 0,C 180,E1 25725.646,E2 25725.646} C_VEL
LIN {X 0,Y 536.453,Z 295.665,A -85,B 0,C 180,E1 25722.426,E2 25722.426} C_VEL
LIN {X 0,Y 536.399,Z 295.661,A -85,B 0,C 180,E1 25719.143,E2 25719.143} C_VEL
LIN {X 0,Y 536.427,Z 295.655,A -85,B 0,C 180,E1 25715.791,E2 25715.791} C_VEL
LIN {X 0,Y 536.442,Z 295.665,A -85,B 0,C 180,E1 25712.521,E2 25712.521} C_VEL
LIN {X 0,Y 536.408,Z 295.662,A -85,B 0,C 180,E1 25709.235,E2 25709.235} C_VEL
LIN {X 0,Y 536.462,Z 295.658,A -85,B 0,C 180,E1 25706.003,E2 25706.003} C_VEL
LIN {X 0,Y 536.42,Z 295.66,A -85,B 0,C 180,E1 25705.427,E2 25705.427} C_VEL
LIN {X 0,Y 535.423,Z 295.79,A -85,B 0,C 180,E1 25704.605,E2 25704.605} C_VEL
LIN {X 0,Y 528.977,Z 296.593,A -85,B 0,C 180,E1 25702.234,E2 25702.234} C_VEL
LIN {X 0,Y 528.507,Z 296.648,A -85,B 0,C 180,E1 25701.691,E2 25701.691} C_VEL
LIN {X 0,Y 528.517,Z 296.649,A -85,B 0,C 180,E1 25698.353,E2 25698.353} C_VEL
LIN {X 0,Y 528.483,Z 296.646,A -85,B 0,C 180,E1 25694.961,E2 25694.961} C_VEL
LIN {X 0,Y 528.518,Z 296.65,A -85,B 0,C 180,E1 25691.606,E2 25691.606} C_VEL
LIN {X 0,Y 528.523,Z 296.635,A -85,B 0,C 180,E1 25688.214,E2 25688.214} C_VEL
LIN {X 0,Y 528.49,Z 296.642,A -85,B 0,C 180,E1 25684.805,E2 25684.805} C_VEL
LIN {X 0,Y 528.511,Z 296.637,A -85,B 0,C 180,E1 25681.348,E2 25681.348} C_VEL
LIN {X 0,Y 528.551,Z 296.858,A -85,B 0,C 180,E1 25680.242,E2 25680.242} C_VEL
LIN {X 0,Y 534.193,Z 314.111,A -85,B 0,C 180,E1 25678.021,E2 25678.021} C_VEL
LIN {X 0,Y 533.42,Z 336.395,A -85,B 0,C 180,E1 25675.877,E2 25675.877} C_VEL
LIN {X 0,Y 535.67,Z 347.817,A -85,B 0,C 180,E1 25675.564,E2 25675.564} C_VEL
LIN {X 0,Y 534.4,Z 545.275,A -85,B 0,C 180,E1 25672.802,E2 25672.802} C_VEL
LIN {X 0,Y 534.083,Z 564.213,A -85,B 0,C 180,E1 25672.332,E2 25672.332} C_VEL
LIN {X 0,Y 533.546,Z 582.504,A -85,B 0,C 180,E1 25671.664,E2 25671.664} C_VEL
LIN {X 0,Y 532.91,Z 599.652,A -85,B 0,C 180,E1 25670.826,E2 25670.826} C_VEL
LIN {X 0,Y 532.155,Z 615.873,A -85,B 0,C 180,E1 25669.824,E2 25669.824} C_VEL
LIN {X 0,Y 531.335,Z 631.837,A -85,B 0,C 180,E1 25668.6,E2 25668.6} C_VEL
LIN {X 0,Y 530.562,Z 646.088,A -85,B 0,C 180,E1 25667.271,E2 25667.271} C_VEL
LIN {X 0,Y 529.803,Z 659.701,A -85,B 0,C 180,E1 25665.742,E2 25665.742} C_VEL
LIN {X 0,Y 529.169,Z 671.804,A -85,B 0,C 180,E1 25664.107,E2 25664.107} C_VEL
LIN {X 0,Y 528.672,Z 682.608,A -85,B 0,C 180,E1 25662.34,E2 25662.34} C_VEL
LIN {X 0,Y 528.292,Z 691.95,A -85,B 0,C 180,E1 25660.468,E2 25660.468} C_VEL
LIN {X 0,Y 528.065,Z 699.796,A -85,B 0,C 180,E1 25658.493,E2 25658.493} C_VEL
LIN {X 0,Y 527.955,Z 706.594,A -85,B 0,C 180,E1 25656.306,E2 25656.306} C_VEL
LIN {X 0,Y 527.924,Z 710.997,A -85,B 0,C 180,E1 25654.345,E2 25654.345} C_VEL
LIN {X 0,Y 527.911,Z 713.744,A -85,B 0,C 180,E1 25652.388,E2 25652.388} C_VEL
LIN {X 0,Y 527.909,Z 714.927,A -85,B 0,C 180,E1 25650.326,E2 25650.326} C_VEL
LIN {X 0,Y 527.913,Z 714.374,A -85,B 0,C 180,E1 25648.264,E2 25648.264} C_VEL
LIN {X 0,Y 527.914,Z 712.226,A -85,B 0,C 180,E1 25646.308,E2 25646.308} C_VEL
LIN {X 0,Y 527.937,Z 708.455,A -85,B 0,C 180,E1 25644.348,E2 25644.348} C_VEL
LIN {X 0,Y 528.008,Z 702.639,A -85,B 0,C 180,E1 25642.274,E2 25642.274} C_VEL
LIN {X 0,Y 528.172,Z 695.607,A -85,B 0,C 180,E1 25640.301,E2 25640.301} C_VEL
LIN {X 0,Y 528.475,Z 687.161,A -85,B 0,C 180,E1 25638.431,E2 25638.431} C_VEL
LIN {X 0,Y 528.915,Z 677.344,A -85,B 0,C 180,E1 25636.666,E2 25636.666} C_VEL
LIN {X 0,Y 529.452,Z 666.189,A -85,B 0,C 180,E1 25635.006,E2 25635.006} C_VEL
LIN {X 0,Y 530.138,Z 653.641,A -85,B 0,C 180,E1 25633.454,E2 25633.454} C_VEL
LIN {X 0,Y 530.911,Z 639.573,A -85,B 0,C 180,E1 25632.002,E2 25632.002} C_VEL
LIN {X 0,Y 531.708,Z 624.712,A -85,B 0,C 180,E1 25630.734,E2 25630.734} C_VEL
LIN {X 0,Y 532.497,Z 608.695,A -85,B 0,C 180,E1 25629.617,E2 25629.617} C_VEL
LIN {X 0,Y 533.226,Z 591.689,A -85,B 0,C 180,E1 25628.669,E2 25628.669} C_VEL
LIN {X 0,Y 533.817,Z 574.117,A -85,B 0,C 180,E1 25627.914,E2 25627.914} C_VEL
LIN {X 0,Y 534.248,Z 555.617,A -85,B 0,C 180,E1 25627.338,E2 25627.338} C_VEL
LIN {X 0,Y 534.478,Z 536.527,A -85,B 0,C 180,E1 25626.962,E2 25626.962} C_VEL
LIN {X 0,Y 535.554,Z 346.222,A -85,B 0,C 180,E1 25624.316,E2 25624.316} C_VEL
LIN {X 0,Y 533.396,Z 336.077,A -85,B 0,C 180,E1 25624.011,E2 25624.011} C_VEL
LIN {X 0,Y 534.104,Z 313.814,A -85,B 0,C 180,E1 25621.852,E2 25621.852} C_VEL
LIN {X 0,Y 528.55,Z 296.845,A -85,B 0,C 180,E1 25619.664,E2 25619.664} C_VEL
LIN {X 0,Y 528.521,Z 296.638,A -85,B 0,C 180,E1 25616.208,E2 25616.208} C_VEL
LIN {X 0,Y 528.499,Z 296.648,A -85,B 0,C 180,E1 25612.796,E2 25612.796} C_VEL
LIN {X 0,Y 528.496,Z 296.654,A -85,B 0,C 180,E1 25609.256,E2 25609.256} C_VEL
LIN {X 0,Y 528.523,Z 296.631,A -85,B 0,C 180,E1 25605.807,E2 25605.807} C_VEL
LIN {X 0,Y 528.504,Z 296.649,A -85,B 0,C 180,E1 25602.455,E2 25602.455} C_VEL
LIN {X 0,Y 528.485,Z 296.651,A -85,B 0,C 180,E1 25599.051,E2 25599.051} C_VEL
LIN {X 0,Y 528.522,Z 296.654,A -85,B 0,C 180,E1 25595.639,E2 25595.639} C_VEL
LIN {X 0,Y 528.503,Z 296.648,A -85,B 0,C 180,E1 25592.243,E2 25592.243} C_VEL
LIN {X 0,Y 528.475,Z 296.65,A -85,B 0,C 180,E1 25588.97,E2 25588.97} C_VEL
LIN {X 0,Y 528.525,Z 296.647,A -85,B 0,C 180,E1 25585.672,E2 25585.672} C_VEL
LIN {X 0,Y 528.48,Z 296.652,A -85,B 0,C 180,E1 25582.311,E2 25582.311} C_VEL
LIN {X 0,Y 528.463,Z 296.65,A -85,B 0,C 180,E1 25578.877,E2 25578.877} C_VEL
LIN {X 0,Y 528.522,Z 296.648,A -85,B 0,C 180,E1 25575.583,E2 25575.583} C_VEL
LIN {X 0,Y 528.46,Z 296.652,A -85,B 0,C 180,E1 25572.345,E2 25572.345} C_VEL
LIN {X 0,Y 528.455,Z 296.645,A -85,B 0,C 180,E1 25568.816,E2 25568.816} C_VEL
LIN {X 0,Y 528.515,Z 296.655,A -85,B 0,C 180,E1 25565.537,E2 25565.537} C_VEL
LIN {X 0,Y 528.448,Z 296.647,A -85,B 0,C 180,E1 25562.277,E2 25562.277} C_VEL
LIN {X 0,Y 528.449,Z 296.652,A -85,B 0,C 180,E1 25558.808,E2 25558.808} C_VEL
LIN {X 0,Y 528.507,Z 296.65,A -85,B 0,C 180,E1 25555.545,E2 25555.545} C_VEL
LIN {X 0,Y 528.45,Z 296.649,A -85,B 0,C 180,E1 25552.28,E2 25552.28} C_VEL
LIN {X 0,Y 528.473,Z 296.653,A -85,B 0,C 180,E1 25548.873,E2 25548.873} C_VEL
LIN {X 0,Y 528.501,Z 296.646,A -85,B 0,C 180,E1 25545.607,E2 25545.607} C_VEL
LIN {X 0,Y 528.46,Z 296.65,A -85,B 0,C 180,E1 25542.379,E2 25542.379} C_VEL
LIN {X 0,Y 528.512,Z 296.65,A -85,B 0,C 180,E1 25539.05,E2 25539.05} C_VEL
LIN {X 0,Y 528.486,Z 296.65,A -85,B 0,C 180,E1 25535.767,E2 25535.767} C_VEL
LIN {X 0,Y 528.472,Z 296.648,A -85,B 0,C 180,E1 25532.385,E2 25532.385} C_VEL
LIN {X 0,Y 528.524,Z 296.646,A -85,B 0,C 180,E1 25529.032,E2 25529.032} C_VEL
LIN {X 0,Y 528.493,Z 296.649,A -85,B 0,C 180,E1 25525.682,E2 25525.682} C_VEL
LIN {X 0,Y 528.482,Z 296.647,A -85,B 0,C 180,E1 25522.261,E2 25522.261} C_VEL
LIN {X 0,Y 528.528,Z 296.63,A -85,B 0,C 180,E1 25518.971,E2 25518.971} C_VEL
LIN {X 0,Y 528.51,Z 296.654,A -85,B 0,C 180,E1 25515.496,E2 25515.496} C_VEL
LIN {X 0,Y 528.491,Z 296.653,A -85,B 0,C 180,E1 25512.045,E2 25512.045} C_VEL
LIN {X 0,Y 528.527,Z 296.642,A -85,B 0,C 180,E1 25508.767,E2 25508.767} C_VEL
LIN {X 0,Y 528.542,Z 296.967,A -85,B 0,C 180,E1 25508.178,E2 25508.178} C_VEL
LIN {X 0,Y 530.603,Z 302.33,A -85,B 0,C 180,E1 25507.627,E2 25507.627} C_VEL
LIN {X 0,Y 537.847,Z 320.134,A -85,B 0,C 180,E1 25505.975,E2 25505.975} C_VEL
LIN {X 0,Y 536.51,Z 373.681,A -85,B 0,C 180,E1 25502.713,E2 25502.713} C_VEL
LIN {X 0,Y 536.214,Z 390.662,A -85,B 0,C 180,E1 25501.726,E2 25501.726} C_VEL
LIN {X 0,Y 537.859,Z 403.647,A -85,B 0,C 180,E1 25501.434,E2 25501.434} C_VEL
LIN {X 0,Y 536.406,Z 594.787,A -85,B 0,C 180,E1 25498.683,E2 25498.683} C_VEL
LIN {X 0,Y 535.833,Z 654.415,A -85,B 0,C 180,E1 25497.791,E2 25497.791} C_VEL
LIN {X 0,Y 535.306,Z 675.429,A -85,B 0,C 180,E1 25497.273,E2 25497.273} C_VEL
LIN {X 0,Y 534.649,Z 695.21,A -85,B 0,C 180,E1 25496.581,E2 25496.581} C_VEL
LIN {X 0,Y 533.887,Z 714.635,A -85,B 0,C 180,E1 25495.698,E2 25495.698} C_VEL
LIN {X 0,Y 533.019,Z 733.838,A -85,B 0,C 180,E1 25494.609,E2 25494.609} C_VEL
LIN {X 0,Y 532.156,Z 751.982,A -85,B 0,C 180,E1 25493.355,E2 25493.355} C_VEL
LIN {X 0,Y 531.341,Z 768.574,A -85,B 0,C 180,E1 25491.991,E2 25491.991} C_VEL
LIN {X 0,Y 530.496,Z 785.443,A -85,B 0,C 180,E1 25490.341,E2 25490.341} C_VEL
LIN {X 0,Y 529.771,Z 800.448,A -85,B 0,C 180,E1 25488.599,E2 25488.599} C_VEL
LIN {X 0,Y 529.181,Z 813.584,A -85,B 0,C 180,E1 25486.803,E2 25486.803} C_VEL
LIN {X 0,Y 528.719,Z 825.381,A -85,B 0,C 180,E1 25484.903,E2 25484.903} C_VEL
LIN {X 0,Y 528.359,Z 836.336,A -85,B 0,C 180,E1 25482.791,E2 25482.791} C_VEL
LIN {X 0,Y 528.139,Z 845.251,A -85,B 0,C 180,E1 25480.692,E2 25480.692} C_VEL
LIN {X 0,Y 528.009,Z 852.377,A -85,B 0,C 180,E1 25478.603,E2 25478.603} C_VEL
LIN {X 0,Y 527.937,Z 858.005,A -85,B 0,C 180,E1 25476.415,E2 25476.415} C_VEL
LIN {X 0,Y 527.911,Z 861.929,A -85,B 0,C 180,E1 25474.236,E2 25474.236} C_VEL
LIN {X 0,Y 527.911,Z 864.306,A -85,B 0,C 180,E1 25471.954,E2 25471.954} C_VEL
LIN {X 0,Y 527.906,Z 864.962,A -85,B 0,C 180,E1 25469.783,E2 25469.783} C_VEL
LIN {X 0,Y 527.902,Z 864.033,A -85,B 0,C 180,E1 25467.612,E2 25467.612} C_VEL
LIN {X 0,Y 527.911,Z 861.449,A -85,B 0,C 180,E1 25465.438,E2 25465.438} C_VEL
LIN {X 0,Y 527.952,Z 857.245,A -85,B 0,C 180,E1 25463.257,E2 25463.257} C_VEL
LIN {X 0,Y 528.024,Z 851.327,A -85,B 0,C 180,E1 25461.068,E2 25461.068} C_VEL
LIN {X 0,Y 528.162,Z 844.013,A -85,B 0,C 180,E1 25458.977,E2 25458.977} C_VEL
LIN {X 0,Y 528.408,Z 834.783,A -85,B 0,C 180,E1 25456.876,E2 25456.876} C_VEL
LIN {X 0,Y 528.767,Z 824.109,A -85,B 0,C 180,E1 25454.874,E2 25454.874} C_VEL
LIN {X 0,Y 529.252,Z 811.725,A -85,B 0,C 180,E1 25452.926,E2 25452.926} C_VEL
LIN {X 0,Y 529.883,Z 797.67,A -85,B 0,C 180,E1 25451.062,E2 25451.062} C_VEL
LIN {X 0,Y 530.612,Z 782.615,A -85,B 0,C 180,E1 25449.368,E2 25449.368} C_VEL
LIN {X 0,Y 531.432,Z 766.62,A -85,B 0,C 180,E1 25447.839,E2 25447.839} C_VEL
LIN {X 0,Y 532.325,Z 748.992,A -85,B 0,C 180,E1 25446.418,E2 25446.418} C_VEL
LIN {X 0,Y 533.204,Z 730.23,A -85,B 0,C 180,E1 25445.164,E2 25445.164} C_VEL
LIN {X 0,Y 534.017,Z 711.348,A -85,B 0,C 180,E1 25444.136,E2 25444.136} C_VEL
LIN {X 0,Y 534.758,Z 692.224,A -85,B 0,C 180,E1 25443.304,E2 25443.304} C_VEL
LIN {X 0,Y 535.382,Z 671.626,A -85,B 0,C 180,E1 25442.621,E2 25442.621} C_VEL
LIN {X 0,Y 535.881,Z 651.072,A -85,B 0,C 180,E1 25442.149,E2 25442.149} C_VEL
LIN {X 0,Y 537.542,Z 449.728,A -85,B 0,C 180,E1 25439.224,E2 25439.224} C_VEL
LIN {X 0,Y 537.667,Z 400.554,A -85,B 0,C 180,E1 25438.508,E2 25438.508} C_VEL
LIN {X 0,Y 536.131,Z 389.177,A -85,B 0,C 180,E1 25438.215,E2 25438.215} C_VEL
LIN {X 0,Y 537.478,Z 334.555,A -85,B 0,C 180,E1 25434.914,E2 25434.914} C_VEL
LIN {X 0,Y 537.765,Z 319.473,A -85,B 0,C 180,E1 25433.977,E2 25433.977} C_VEL
LIN {X 0,Y 528.559,Z 297.071,A -85,B 0,C 180,E1 25431.843,E2 25431.843} C_VEL
LIN {X 0,Y 528.513,Z 296.65,A -85,B 0,C 180,E1 25431.509,E2 25431.509} C_VEL
LIN {X 0,Y 528.491,Z 296.654,A -85,B 0,C 180,E1 25428.101,E2 25428.101} C_VEL
LIN {X 0,Y 528.521,Z 296.649,A -85,B 0,C 180,E1 25424.659,E2 25424.659} C_VEL
LIN {X 0,Y 528.524,Z 296.628,A -85,B 0,C 180,E1 25421.173,E2 25421.173} C_VEL
LIN {X 0,Y 528.482,Z 296.647,A -85,B 0,C 180,E1 25417.806,E2 25417.806} C_VEL
LIN {X 0,Y 528.504,Z 296.645,A -85,B 0,C 180,E1 25414.429,E2 25414.429} C_VEL
LIN {X 0,Y 528.514,Z 296.647,A -85,B 0,C 180,E1 25411.095,E2 25411.095} C_VEL
LIN {X 0,Y 528.473,Z 296.648,A -85,B 0,C 180,E1 25407.738,E2 25407.738} C_VEL
LIN {X 0,Y 528.5,Z 296.651,A -85,B 0,C 180,E1 25404.357,E2 25404.357} C_VEL
LIN {X 0,Y 528.492,Z 296.651,A -85,B 0,C 180,E1 25401.143,E2 25401.143} C_VEL
LIN {X 0,Y 528.463,Z 296.65,A -85,B 0,C 180,E1 25397.735,E2 25397.735} C_VEL
LIN {X 0,Y 528.505,Z 296.646,A -85,B 0,C 180,E1 25394.395,E2 25394.395} C_VEL
LIN {X 0,Y 528.474,Z 296.652,A -85,B 0,C 180,E1 25391.127,E2 25391.127} C_VEL
LIN {X 0,Y 528.454,Z 296.649,A -85,B 0,C 180,E1 25387.72,E2 25387.72} C_VEL
LIN {X 0,Y 528.511,Z 296.651,A -85,B 0,C 180,E1 25384.448,E2 25384.448} C_VEL
LIN {X 0,Y 528.453,Z 296.652,A -85,B 0,C 180,E1 25381.192,E2 25381.192} C_VEL
LIN {X 0,Y 528.445,Z 296.648,A -85,B 0,C 180,E1 25377.723,E2 25377.723} C_VEL
LIN {X 0,Y 528.509,Z 296.654,A -85,B 0,C 180,E1 25374.463,E2 25374.463} C_VEL
LIN {X 0,Y 528.446,Z 296.645,A -85,B 0,C 180,E1 25371.294,E2 25371.294} C_VEL
LIN {X 0,Y 528.481,Z 296.652,A -85,B 0,C 180,E1 25367.988,E2 25367.988} C_VEL
LIN {X 0,Y 528.469,Z 296.647,A -85,B 0,C 180,E1 25364.865,E2 25364.865} C_VEL
LIN {X 0,Y 528.46,Z 296.649,A -85,B 0,C 180,E1 25361.419,E2 25361.419} C_VEL
LIN {X 0,Y 528.519,Z 296.651,A -85,B 0,C 180,E1 25358.118,E2 25358.118} C_VEL
LIN {X 0,Y 528.476,Z 296.646,A -85,B 0,C 180,E1 25354.805,E2 25354.805} C_VEL
LIN {X 0,Y 528.471,Z 296.649,A -85,B 0,C 180,E1 25351.385,E2 25351.385} C_VEL
LIN {X 0,Y 528.53,Z 296.651,A -85,B 0,C 180,E1 25348.142,E2 25348.142} C_VEL
LIN {X 0,Y 528.482,Z 296.652,A -85,B 0,C 180,E1 25344.757,E2 25344.757} C_VEL
LIN {X 0,Y 528.507,Z 296.648,A -85,B 0,C 180,E1 25341.691,E2 25341.691} C_VEL
LIN {X 0,Y 527.481,Z 296.777,A -85,B 0,C 180,E1 25340.857,E2 25340.857} C_VEL
LIN {X 0,Y 521.034,Z 297.584,A -85,B 0,C 180,E1 25338.45,E2 25338.45} C_VEL
LIN {X 0,Y 520.588,Z 297.638,A -85,B 0,C 180,E1 25337.9,E2 25337.9} C_VEL
LIN {X 0,Y 520.562,Z 297.625,A -85,B 0,C 180,E1 25334.511,E2 25334.511} C_VEL
LIN {X 0,Y 520.548,Z 297.642,A -85,B 0,C 180,E1 25331.063,E2 25331.063} C_VEL
LIN {X 0,Y 520.582,Z 297.628,A -85,B 0,C 180,E1 25327.644,E2 25327.644} C_VEL
LIN {X 0,Y 520.583,Z 297.622,A -85,B 0,C 180,E1 25324.126,E2 25324.126} C_VEL
LIN {X 0,Y 520.579,Z 297.806,A -85,B 0,C 180,E1 25320.755,E2 25320.755} C_VEL
LIN {X 0,Y 526.918,Z 316.989,A -85,B 0,C 180,E1 25318.234,E2 25318.234} C_VEL
LIN {X 0,Y 526.229,Z 337.08,A -85,B 0,C 180,E1 25316.302,E2 25316.302} C_VEL
LIN {X 0,Y 528.672,Z 349.224,A -85,B 0,C 180,E1 25315.966,E2 25315.966} C_VEL
LIN {X 0,Y 527.369,Z 546.9,A -85,B 0,C 180,E1 25313.192,E2 25313.192} C_VEL
LIN {X 0,Y 527.036,Z 565.736,A -85,B 0,C 180,E1 25312.713,E2 25312.713} C_VEL
LIN {X 0,Y 526.49,Z 583.327,A -85,B 0,C 180,E1 25312.064,E2 25312.064} C_VEL
LIN {X 0,Y 525.813,Z 600.136,A -85,B 0,C 180,E1 25311.238,E2 25311.238} C_VEL
LIN {X 0,Y 524.982,Z 616.458,A -85,B 0,C 180,E1 25310.223,E2 25310.223} C_VEL
LIN {X 0,Y 524.076,Z 632.536,A -85,B 0,C 180,E1 25308.983,E2 25308.983} C_VEL
LIN {X 0,Y 523.164,Z 647.431,A -85,B 0,C 180,E1 25307.575,E2 25307.575} C_VEL
LIN {X 0,Y 522.291,Z 661.177,A -85,B 0,C 180,E1 25306.001,E2 25306.001} C_VEL
LIN {X 0,Y 521.551,Z 673.351,A -85,B 0,C 180,E1 25304.318,E2 25304.318} C_VEL
LIN {X 0,Y 520.971,Z 684.051,A -85,B 0,C 180,E1 25302.525,E2 25302.525} C_VEL
LIN {X 0,Y 520.525,Z 693.329,A -85,B 0,C 180,E1 25300.626,E2 25300.626} C_VEL
LIN {X 0,Y 520.241,Z 701.12,A -85,B 0,C 180,E1 25298.621,E2 25298.621} C_VEL
LIN {X 0,Y 520.062,Z 707.368,A -85,B 0,C 180,E1 25296.513,E2 25296.513} C_VEL
LIN {X 0,Y 519.972,Z 711.771,A -85,B 0,C 180,E1 25294.411,E2 25294.411} C_VEL
LIN {X 0,Y 519.937,Z 714.447,A -85,B 0,C 180,E1 25292.314,E2 25292.314} C_VEL
LIN {X 0,Y 519.928,Z 715.468,A -85,B 0,C 180,E1 25290.22,E2 25290.22} C_VEL
LIN {X 0,Y 519.935,Z 714.863,A -85,B 0,C 180,E1 25288.127,E2 25288.127} C_VEL
LIN {X 0,Y 519.959,Z 712.615,A -85,B 0,C 180,E1 25286.031,E2 25286.031} C_VEL
LIN {X 0,Y 520.032,Z 708.67,A -85,B 0,C 180,E1 25283.93,E2 25283.93} C_VEL
LIN {X 0,Y 520.194,Z 702.925,A -85,B 0,C 180,E1 25281.823,E2 25281.823} C_VEL
LIN {X 0,Y 520.44,Z 695.647,A -85,B 0,C 180,E1 25279.82,E2 25279.82} C_VEL
LIN {X 0,Y 520.865,Z 686.322,A -85,B 0,C 180,E1 25277.81,E2 25277.81} C_VEL
LIN {X 0,Y 521.412,Z 675.998,A -85,B 0,C 180,E1 25276.003,E2 25276.003} C_VEL
LIN {X 0,Y 522.09,Z 664.479,A -85,B 0,C 180,E1 25274.334,E2 25274.334} C_VEL
LIN {X 0,Y 522.912,Z 651.395,A -85,B 0,C 180,E1 25272.761,E2 25272.761} C_VEL
LIN {X 0,Y 523.776,Z 637.316,A -85,B 0,C 180,E1 25271.353,E2 25271.353} C_VEL
LIN {X 0,Y 524.663,Z 622.309,A -85,B 0,C 180,E1 25270.113,E2 25270.113} C_VEL
LIN {X 0,Y 525.501,Z 606.44,A -85,B 0,C 180,E1 25269.041,E2 25269.041} C_VEL
LIN {X 0,Y 526.243,Z 589.686,A -85,B 0,C 180,E1 25268.137,E2 25268.137} C_VEL
LIN {X 0,Y 526.854,Z 572.11,A -85,B 0,C 180,E1 25267.411,E2 25267.411} C_VEL
LIN {X 0,Y 527.266,Z 553.957,A -85,B 0,C 180,E1 25266.875,E2 25266.875} C_VEL
LIN {X 0,Y 527.468,Z 534.429,A -85,B 0,C 180,E1 25266.515,E2 25266.515} C_VEL
LIN {X 0,Y 528.54,Z 347.505,A -85,B 0,C 180,E1 25263.91,E2 25263.91} C_VEL
LIN {X 0,Y 526.205,Z 336.939,A -85,B 0,C 180,E1 25263.601,E2 25263.601} C_VEL
LIN {X 0,Y 526.942,Z 317.05,A -85,B 0,C 180,E1 25261.683,E2 25261.683} C_VEL
LIN {X 0,Y 520.582,Z 297.802,A -85,B 0,C 180,E1 25259.15,E2 25259.15} C_VEL
LIN {X 0,Y 520.579,Z 297.622,A -85,B 0,C 180,E1 25255.679,E2 25255.679} C_VEL
LIN {X 0,Y 520.586,Z 297.627,A -85,B 0,C 180,E1 25252.217,E2 25252.217} C_VEL
LIN {X 0,Y 520.556,Z 297.64,A -85,B 0,C 180,E1 25248.792,E2 25248.792} C_VEL
LIN {X 0,Y 520.557,Z 297.627,A -85,B 0,C 180,E1 25245.29,E2 25245.29} C_VEL
LIN {X 0,Y 520.589,Z 297.638,A -85,B 0,C 180,E1 25241.942,E2 25241.942} C_VEL
LIN {X 0,Y 520.551,Z 297.637,A -85,B 0,C 180,E1 25238.581,E2 25238.581} C_VEL
LIN {X 0,Y 520.543,Z 297.639,A -85,B 0,C 180,E1 25235.052,E2 25235.052} C_VEL
LIN {X 0,Y 520.585,Z 297.643,A -85,B 0,C 180,E1 25231.624,E2 25231.624} C_VEL
LIN {X 0,Y 520.552,Z 297.636,A -85,B 0,C 180,E1 25228.323,E2 25228.323} C_VEL
LIN {X 0,Y 520.53,Z 297.633,A -85,B 0,C 180,E1 25224.877,E2 25224.877} C_VEL
LIN {X 0,Y 520.578,Z 297.64,A -85,B 0,C 180,E1 25221.522,E2 25221.522} C_VEL
LIN {X 0,Y 520.538,Z 297.637,A -85,B 0,C 180,E1 25218.246,E2 25218.246} C_VEL
LIN {X 0,Y 520.519,Z 297.634,A -85,B 0,C 180,E1 25214.802,E2 25214.802} C_VEL
LIN {X 0,Y 520.576,Z 297.644,A -85,B 0,C 180,E1 25211.523,E2 25211.523} C_VEL
LIN {X 0,Y 520.524,Z 297.632,A -85,B 0,C 180,E1 25208.172,E2 25208.172} C_VEL
LIN {X 0,Y 520.51,Z 297.642,A -85,B 0,C 180,E1 25204.738,E2 25204.738} C_VEL
LIN {X 0,Y 520.568,Z 297.638,A -85,B 0,C 180,E1 25201.431,E2 25201.431} C_VEL
LIN {X 0,Y 520.513,Z 297.64,A -85,B 0,C 180,E1 25198.129,E2 25198.129} C_VEL
LIN {X 0,Y 520.513,Z 297.643,A -85,B 0,C 180,E1 25194.71,E2 25194.71} C_VEL
LIN {X 0,Y 520.573,Z 297.633,A -85,B 0,C 180,E1 25191.495,E2 25191.495} C_VEL
LIN {X 0,Y 520.52,Z 297.643,A -85,B 0,C 180,E1 25188.139,E2 25188.139} C_VEL
LIN {X 0,Y 520.526,Z 297.642,A -85,B 0,C 180,E1 25184.629,E2 25184.629} C_VEL
LIN {X 0,Y 520.583,Z 297.634,A -85,B 0,C 180,E1 25181.292,E2 25181.292} C_VEL
LIN {X 0,Y 520.532,Z 297.642,A -85,B 0,C 180,E1 25178.003,E2 25178.003} C_VEL
LIN {X 0,Y 520.536,Z 297.641,A -85,B 0,C 180,E1 25174.516,E2 25174.516} C_VEL
LIN {X 0,Y 520.589,Z 297.64,A -85,B 0,C 180,E1 25171.137,E2 25171.137} C_VEL
LIN {X 0,Y 520.551,Z 297.641,A -85,B 0,C 180,E1 25167.726,E2 25167.726} C_VEL
LIN {X 0,Y 520.539,Z 297.621,A -85,B 0,C 180,E1 25164.273,E2 25164.273} C_VEL
LIN {X 0,Y 520.589,Z 297.637,A -85,B 0,C 180,E1 25160.888,E2 25160.888} C_VEL
LIN {X 0,Y 520.572,Z 297.622,A -85,B 0,C 180,E1 25157.462,E2 25157.462} C_VEL
LIN {X 0,Y 520.548,Z 297.626,A -85,B 0,C 180,E1 25154.051,E2 25154.051} C_VEL
LIN {X 0,Y 520.584,Z 297.625,A -85,B 0,C 180,E1 25150.623,E2 25150.623} C_VEL
LIN {X 0,Y 520.602,Z 297.735,A -85,B 0,C 180,E1 25148.762,E2 25148.762} C_VEL
LIN {X 0,Y 520.932,Z 299.194,A -85,B 0,C 180,E1 25148.552,E2 25148.552} C_VEL
LIN {X 0,Y 530.761,Z 322.797,A -85,B 0,C 180,E1 25146.278,E2 25146.278} C_VEL
LIN {X 0,Y 529.242,Z 376.53,A -85,B 0,C 180,E1 25142.962,E2 25142.962} C_VEL
LIN {X 0,Y 528.955,Z 390.189,A -85,B 0,C 180,E1 25142.157,E2 25142.157} C_VEL
LIN {X 0,Y 530.787,Z 404.692,A -85,B 0,C 180,E1 25141.824,E2 25141.824} C_VEL
LIN {X 0,Y 529.1,Z 621.359,A -85,B 0,C 180,E1 25138.704,E2 25138.704} C_VEL
LIN {X 0,Y 528.723,Z 655.388,A -85,B 0,C 180,E1 25138.175,E2 25138.175} C_VEL
LIN {X 0,Y 528.15,Z 676.307,A -85,B 0,C 180,E1 25137.647,E2 25137.647} C_VEL
LIN {X 0,Y 527.422,Z 696.021,A -85,B 0,C 180,E1 25136.941,E2 25136.941} C_VEL
LIN {X 0,Y 526.599,Z 714.743,A -85,B 0,C 180,E1 25136.074,E2 25136.074} C_VEL
LIN {X 0,Y 525.642,Z 733.835,A -85,B 0,C 180,E1 25134.978,E2 25134.978} C_VEL
LIN {X 0,Y 524.69,Z 751.979,A -85,B 0,C 180,E1 25133.708,E2 25133.708} C_VEL
LIN {X 0,Y 523.737,Z 769.18,A -85,B 0,C 180,E1 25132.268,E2 25132.268} C_VEL
LIN {X 0,Y 522.831,Z 785.377,A -85,B 0,C 180,E1 25130.66,E2 25130.66} C_VEL
LIN {X 0,Y 522.011,Z 800.505,A -85,B 0,C 180,E1 25128.879,E2 25128.879} C_VEL
LIN {X 0,Y 521.319,Z 814.353,A -85,B 0,C 180,E1 25126.949,E2 25126.949} C_VEL
LIN {X 0,Y 520.807,Z 826.015,A -85,B 0,C 180,E1 25125.021,E2 25125.021} C_VEL
LIN {X 0,Y 520.406,Z 836.85,A -85,B 0,C 180,E1 25122.877,E2 25122.877} C_VEL
LIN {X 0,Y 520.152,Z 846.063,A -85,B 0,C 180,E1 25120.634,E2 25120.634} C_VEL
LIN {X 0,Y 520.008,Z 853.292,A -85,B 0,C 180,E1 25118.403,E2 25118.403} C_VEL
LIN {X 0,Y 519.941,Z 858.728,A -85,B 0,C 180,E1 25116.182,E2 25116.182} C_VEL
LIN {X 0,Y 519.916,Z 862.403,A -85,B 0,C 180,E1 25113.97,E2 25113.97} C_VEL
LIN {X 0,Y 519.907,Z 864.442,A -85,B 0,C 180,E1 25111.763,E2 25111.763} C_VEL
LIN {X 0,Y 519.9,Z 864.895,A -85,B 0,C 180,E1 25109.449,E2 25109.449} C_VEL
LIN {X 0,Y 519.912,Z 863.73,A -85,B 0,C 180,E1 25107.244,E2 25107.244} C_VEL
LIN {X 0,Y 519.93,Z 860.86,A -85,B 0,C 180,E1 25104.967,E2 25104.967} C_VEL
LIN {X 0,Y 519.971,Z 856.228,A -85,B 0,C 180,E1 25102.709,E2 25102.709} C_VEL
LIN {X 0,Y 520.067,Z 850.267,A -85,B 0,C 180,E1 25100.595,E2 25100.595} C_VEL
LIN {X 0,Y 520.251,Z 842.178,A -85,B 0,C 180,E1 25098.358,E2 25098.358} C_VEL
LIN {X 0,Y 520.563,Z 832.564,A -85,B 0,C 180,E1 25096.222,E2 25096.222} C_VEL
LIN {X 0,Y 521.001,Z 821.489,A -85,B 0,C 180,E1 25094.187,E2 25094.187} C_VEL
LIN {X 0,Y 521.587,Z 808.952,A -85,B 0,C 180,E1 25092.255,E2 25092.255} C_VEL
LIN {X 0,Y 522.304,Z 794.891,A -85,B 0,C 180,E1 25090.428,E2 25090.428} C_VEL
LIN {X 0,Y 523.127,Z 779.839,A -85,B 0,C 180,E1 25088.766,E2 25088.766} C_VEL
LIN {X 0,Y 524.048,Z 763.286,A -85,B 0,C 180,E1 25087.213,E2 25087.213} C_VEL
LIN {X 0,Y 525.059,Z 745.028,A -85,B 0,C 180,E1 25085.779,E2 25085.779} C_VEL
LIN {X 0,Y 526.045,Z 726.288,A -85,B 0,C 180,E1 25084.561,E2 25084.561} C_VEL
LIN {X 0,Y 526.947,Z 707.342,A -85,B 0,C 180,E1 25083.557,E2 25083.557} C_VEL
LIN {X 0,Y 527.74,Z 687.885,A -85,B 0,C 180,E1 25082.741,E2 25082.741} C_VEL
LIN {X 0,Y 528.402,Z 667.723,A -85,B 0,C 180,E1 25082.114,E2 25082.114} C_VEL
LIN {X 0,Y 528.851,Z 647.19,A -85,B 0,C 180,E1 25081.676,E2 25081.676} C_VEL
LIN {X 0,Y 530.711,Z 411.968,A -85,B 0,C 180,E1 25078.284,E2 25078.284} C_VEL
LIN {X 0,Y 530.565,Z 401.444,A -85,B 0,C 180,E1 25078.113,E2 25078.113} C_VEL
LIN {X 0,Y 528.878,Z 388.739,A -85,B 0,C 180,E1 25077.784,E2 25077.784} C_VEL
LIN {X 0,Y 530.436,Z 334.357,A -85,B 0,C 180,E1 25074.444,E2 25074.444} C_VEL
LIN {X 0,Y 530.669,Z 322.582,A -85,B 0,C 180,E1 25073.701,E2 25073.701} C_VEL
LIN {X 0,Y 520.651,Z 298.067,A -85,B 0,C 180,E1 25071.319,E2 25071.319} C_VEL
LIN {X 0,Y 520.584,Z 297.624,A -85,B 0,C 180,E1 25070.953,E2 25070.953} C_VEL
LIN {X 0,Y 520.568,Z 297.635,A -85,B 0,C 180,E1 25067.523,E2 25067.523} C_VEL
LIN {X 0,Y 520.549,Z 297.643,A -85,B 0,C 180,E1 25064.053,E2 25064.053} C_VEL
LIN {X 0,Y 520.582,Z 297.625,A -85,B 0,C 180,E1 25060.624,E2 25060.624} C_VEL
LIN {X 0,Y 520.581,Z 297.626,A -85,B 0,C 180,E1 25057.151,E2 25057.151} C_VEL
LIN {X 0,Y 520.541,Z 297.64,A -85,B 0,C 180,E1 25053.718,E2 25053.718} C_VEL
LIN {X 0,Y 520.55,Z 297.644,A -85,B 0,C 180,E1 25050.214,E2 25050.214} C_VEL
LIN {X 0,Y 520.581,Z 297.634,A -85,B 0,C 180,E1 25046.954,E2 25046.954} C_VEL
LIN {X 0,Y 520.531,Z 297.637,A -85,B 0,C 180,E1 25043.621,E2 25043.621} C_VEL
LIN {X 0,Y 520.549,Z 297.641,A -85,B 0,C 180,E1 25040.227,E2 25040.227} C_VEL
LIN {X 0,Y 520.572,Z 297.637,A -85,B 0,C 180,E1 25036.859,E2 25036.859} C_VEL
LIN {X 0,Y 520.519,Z 297.632,A -85,B 0,C 180,E1 25033.553,E2 25033.553} C_VEL
LIN {X 0,Y 520.544,Z 297.641,A -85,B 0,C 180,E1 25030.178,E2 25030.178} C_VEL
LIN {X 0,Y 520.542,Z 297.637,A -85,B 0,C 180,E1 25026.95,E2 25026.95} C_VEL
LIN {X 0,Y 520.51,Z 297.638,A -85,B 0,C 180,E1 25023.634,E2 25023.634} C_VEL
LIN {X 0,Y 520.563,Z 297.644,A -85,B 0,C 180,E1 25020.33,E2 25020.33} C_VEL
LIN {X 0,Y 520.516,Z 297.636,A -85,B 0,C 180,E1 25017.027,E2 25017.027} C_VEL
LIN {X 0,Y 520.508,Z 297.643,A -85,B 0,C 180,E1 25013.603,E2 25013.603} C_VEL
LIN {X 0,Y 520.572,Z 297.635,A -85,B 0,C 180,E1 25010.381,E2 25010.381} C_VEL
LIN {X 0,Y 520.516,Z 297.642,A -85,B 0,C 180,E1 25007.125,E2 25007.125} C_VEL
LIN {X 0,Y 520.524,Z 297.642,A -85,B 0,C 180,E1 25003.598,E2 25003.598} C_VEL
LIN {X 0,Y 520.581,Z 297.632,A -85,B 0,C 180,E1 25000.236,E2 25000.236} C_VEL
LIN {X 0,Y 520.531,Z 297.643,A -85,B 0,C 180,E1 24996.93,E2 24996.93} C_VEL
LIN {X 0,Y 520.531,Z 297.641,A -85,B 0,C 180,E1 24993.413,E2 24993.413} C_VEL
LIN {X 0,Y 520.591,Z 297.634,A -85,B 0,C 180,E1 24990.042,E2 24990.042} C_VEL
LIN {X 0,Y 520.551,Z 297.642,A -85,B 0,C 180,E1 24986.669,E2 24986.669} C_VEL
LIN {X 0,Y 520.538,Z 297.641,A -85,B 0,C 180,E1 24983.18,E2 24983.18} C_VEL
LIN {X 0,Y 520.58,Z 297.637,A -85,B 0,C 180,E1 24979.808,E2 24979.808} C_VEL
LIN {X 0,Y 520.588,Z 297.638,A -85,B 0,C 180,E1 24977.9,E2 24977.9} C_VEL
LIN {X 0,Y 519.576,Z 297.762,A -85,B 0,C 180,E1 24977.052,E2 24977.052} C_VEL
LIN {X 0,Y 513.168,Z 298.548,A -85,B 0,C 180,E1 24974.67,E2 24974.67} C_VEL
LIN {X 0,Y 512.646,Z 298.604,A -85,B 0,C 180,E1 24974.05,E2 24974.05} C_VEL
LIN {X 0,Y 512.616,Z 298.634,A -85,B 0,C 180,E1 24970.646,E2 24970.646} C_VEL
LIN {X 0,Y 512.614,Z 298.627,A -85,B 0,C 180,E1 24967.083,E2 24967.083} C_VEL
LIN {X 0,Y 512.644,Z 298.613,A -85,B 0,C 180,E1 24963.61,E2 24963.61} C_VEL
LIN {X 0,Y 512.665,Z 298.875,A -85,B 0,C 180,E1 24961.25,E2 24961.25} C_VEL
LIN {X 0,Y 519.539,Z 319.478,A -85,B 0,C 180,E1 24958.507,E2 24958.507} C_VEL
LIN {X 0,Y 519.024,Z 337.459,A -85,B 0,C 180,E1 24956.752,E2 24956.752} C_VEL
LIN {X 0,Y 521.699,Z 350.573,A -85,B 0,C 180,E1 24956.38,E2 24956.38} C_VEL
LIN {X 0,Y 520.375,Z 547.955,A -85,B 0,C 180,E1 24953.604,E2 24953.604} C_VEL
LIN {X 0,Y 520.037,Z 566.771,A -85,B 0,C 180,E1 24953.122,E2 24953.122} C_VEL
LIN {X 0,Y 519.458,Z 584.493,A -85,B 0,C 180,E1 24952.462,E2 24952.462} C_VEL
LIN {X 0,Y 518.708,Z 601.722,A -85,B 0,C 180,E1 24951.602,E2 24951.602} C_VEL
LIN {X 0,Y 517.807,Z 617.966,A -85,B 0,C 180,E1 24950.574,E2 24950.574} C_VEL
LIN {X 0,Y 516.804,Z 633.932,A -85,B 0,C 180,E1 24949.319,E2 24949.319} C_VEL
LIN {X 0,Y 515.83,Z 648.22,A -85,B 0,C 180,E1 24947.95,E2 24947.95} C_VEL
LIN {X 0,Y 514.848,Z 661.999,A -85,B 0,C 180,E1 24946.355,E2 24946.355} C_VEL
LIN {X 0,Y 514.002,Z 674.218,A -85,B 0,C 180,E1 24944.648,E2 24944.648} C_VEL
LIN {X 0,Y 513.328,Z 684.954,A -85,B 0,C 180,E1 24942.829,E2 24942.829} C_VEL
LIN {X 0,Y 512.79,Z 694.248,A -85,B 0,C 180,E1 24940.902,E2 24940.902} C_VEL
LIN {X 0,Y 512.43,Z 702.067,A -85,B 0,C 180,E1 24938.867,E2 24938.867} C_VEL
LIN {X 0,Y 512.211,Z 708.354,A -85,B 0,C 180,E1 24936.726,E2 24936.726} C_VEL
LIN {X 0,Y 512.086,Z 712.811,A -85,B 0,C 180,E1 24934.592,E2 24934.592} C_VEL
LIN {X 0,Y 512.031,Z 715.552,A -85,B 0,C 180,E1 24932.462,E2 24932.462} C_VEL
LIN {X 0,Y 512.018,Z 716.649,A -85,B 0,C 180,E1 24930.336,E2 24930.336} C_VEL
LIN {X 0,Y 512.027,Z 716.132,A -85,B 0,C 180,E1 24928.21,E2 24928.21} C_VEL
LIN {X 0,Y 512.061,Z 713.989,A -85,B 0,C 180,E1 24926.081,E2 24926.081} C_VEL
LIN {X 0,Y 512.153,Z 710.161,A -85,B 0,C 180,E1 24923.949,E2 24923.949} C_VEL
LIN {X 0,Y 512.346,Z 704.552,A -85,B 0,C 180,E1 24921.81,E2 24921.81} C_VEL
LIN {X 0,Y 512.637,Z 697.451,A -85,B 0,C 180,E1 24919.777,E2 24919.777} C_VEL
LIN {X 0,Y 513.133,Z 688.386,A -85,B 0,C 180,E1 24917.738,E2 24917.738} C_VEL
LIN {X 0,Y 513.787,Z 677.664,A -85,B 0,C 180,E1 24915.807,E2 24915.807} C_VEL
LIN {X 0,Y 514.558,Z 666.154,A -85,B 0,C 180,E1 24914.099,E2 24914.099} C_VEL
LIN {X 0,Y 515.475,Z 653.203,A -85,B 0,C 180,E1 24912.504,E2 24912.504} C_VEL
LIN {X 0,Y 516.437,Z 639.312,A -85,B 0,C 180,E1 24911.078,E2 24911.078} C_VEL
LIN {X 0,Y 517.416,Z 624.536,A -85,B 0,C 180,E1 24909.823,E2 24909.823} C_VEL
LIN {X 0,Y 518.326,Z 608.947,A -85,B 0,C 180,E1 24908.737,E2 24908.737} C_VEL
LIN {X 0,Y 519.137,Z 592.552,A -85,B 0,C 180,E1 24907.822,E2 24907.822} C_VEL
LIN {X 0,Y 519.815,Z 574.501,A -85,B 0,C 180,E1 24907.051,E2 24907.051} C_VEL
LIN {X 0,Y 520.26,Z 556.025,A -85,B 0,C 180,E1 24906.487,E2 24906.487} C_VEL
LIN {X 0,Y 520.461,Z 536.725,A -85,B 0,C 180,E1 24906.12,E2 24906.12} C_VEL
LIN {X 0,Y 521.552,Z 348.835,A -85,B 0,C 180,E1 24903.494,E2 24903.494} C_VEL
LIN {X 0,Y 518.981,Z 336.969,A -85,B 0,C 180,E1 24903.127,E2 24903.127} C_VEL
LIN {X 0,Y 519.601,Z 319.667,A -85,B 0,C 180,E1 24901.428,E2 24901.428} C_VEL
LIN {X 0,Y 513.355,Z 301.104,A -85,B 0,C 180,E1 24898.98,E2 24898.98} C_VEL
LIN {X 0,Y 512.658,Z 298.755,A -85,B 0,C 180,E1 24898.619,E2 24898.619} C_VEL
LIN {X 0,Y 512.618,Z 298.615,A -85,B 0,C 180,E1 24895.147,E2 24895.147} C_VEL
LIN {X 0,Y 512.64,Z 298.609,A -85,B 0,C 180,E1 24891.635,E2 24891.635} C_VEL
LIN {X 0,Y 512.65,Z 298.628,A -85,B 0,C 180,E1 24888.163,E2 24888.163} C_VEL
LIN {X 0,Y 512.614,Z 298.622,A -85,B 0,C 180,E1 24884.76,E2 24884.76} C_VEL
LIN {X 0,Y 512.614,Z 298.628,A -85,B 0,C 180,E1 24881.245,E2 24881.245} C_VEL
LIN {X 0,Y 512.65,Z 298.623,A -85,B 0,C 180,E1 24877.826,E2 24877.826} C_VEL
LIN {X 0,Y 512.617,Z 298.625,A -85,B 0,C 180,E1 24874.408,E2 24874.408} C_VEL
LIN {X 0,Y 512.6,Z 298.629,A -85,B 0,C 180,E1 24870.994,E2 24870.994} C_VEL
LIN {X 0,Y 512.646,Z 298.629,A -85,B 0,C 180,E1 24867.658,E2 24867.658} C_VEL
LIN {X 0,Y 512.606,Z 298.62,A -85,B 0,C 180,E1 24864.303,E2 24864.303} C_VEL
LIN {X 0,Y 512.591,Z 298.627,A -85,B 0,C 180,E1 24860.883,E2 24860.883} C_VEL
LIN {X 0,Y 512.633,Z 298.632,A -85,B 0,C 180,E1 24857.48,E2 24857.48} C_VEL
LIN {X 0,Y 512.601,Z 298.621,A -85,B 0,C 180,E1 24854.112,E2 24854.112} C_VEL
LIN {X 0,Y 512.576,Z 298.631,A -85,B 0,C 180,E1 24850.68,E2 24850.68} C_VEL
LIN {X 0,Y 512.612,Z 298.631,A -85,B 0,C 180,E1 24847.284,E2 24847.284} C_VEL
LIN {X 0,Y 512.589,Z 298.631,A -85,B 0,C 180,E1 24844.027,E2 24844.027} C_VEL
LIN {X 0,Y 512.566,Z 298.633,A -85,B 0,C 180,E1 24840.671,E2 24840.671} C_VEL
LIN {X 0,Y 512.628,Z 298.62,A -85,B 0,C 180,E1 24837.429,E2 24837.429} C_VEL
LIN {X 0,Y 512.581,Z 298.632,A -85,B 0,C 180,E1 24834.066,E2 24834.066} C_VEL
LIN {X 0,Y 512.576,Z 298.629,A -85,B 0,C 180,E1 24830.57,E2 24830.57} C_VEL
LIN {X 0,Y 512.632,Z 298.62,A -85,B 0,C 180,E1 24827.211,E2 24827.211} C_VEL
LIN {X 0,Y 512.594,Z 298.632,A -85,B 0,C 180,E1 24823.92,E2 24823.92} C_VEL
LIN {X 0,Y 512.587,Z 298.628,A -85,B 0,C 180,E1 24820.41,E2 24820.41} C_VEL
LIN {X 0,Y 512.637,Z 298.622,A -85,B 0,C 180,E1 24817.04,E2 24817.04} C_VEL
LIN {X 0,Y 512.624,Z 298.629,A -85,B 0,C 180,E1 24813.596,E2 24813.596} C_VEL
LIN {X 0,Y 512.596,Z 298.631,A -85,B 0,C 180,E1 24810.225,E2 24810.225} C_VEL
LIN {X 0,Y 512.63,Z 298.627,A -85,B 0,C 180,E1 24806.795,E2 24806.795} C_VEL
LIN {X 0,Y 512.641,Z 298.604,A -85,B 0,C 180,E1 24803.357,E2 24803.357} C_VEL
LIN {X 0,Y 512.608,Z 298.63,A -85,B 0,C 180,E1 24799.934,E2 24799.934} C_VEL
LIN {X 0,Y 512.624,Z 298.629,A -85,B 0,C 180,E1 24796.487,E2 24796.487} C_VEL
LIN {X 0,Y 512.646,Z 298.61,A -85,B 0,C 180,E1 24793.048,E2 24793.048} C_VEL
LIN {X 0,Y 512.623,Z 298.609,A -85,B 0,C 180,E1 24789.607,E2 24789.607} C_VEL
LIN {X 0,Y 512.684,Z 298.875,A -85,B 0,C 180,E1 24789.264,E2 24789.264} C_VEL
LIN {X 0,Y 514.331,Z 303.21,A -85,B 0,C 180,E1 24788.782,E2 24788.782} C_VEL
LIN {X 0,Y 523.7,Z 325.924,A -85,B 0,C 180,E1 24786.56,E2 24786.56} C_VEL
LIN {X 0,Y 521.975,Z 379.355,A -85,B 0,C 180,E1 24783.218,E2 24783.218} C_VEL
LIN {X 0,Y 521.733,Z 389.76,A -85,B 0,C 180,E1 24782.599,E2 24782.599} C_VEL
LIN {X 0,Y 523.737,Z 405.858,A -85,B 0,C 180,E1 24782.223,E2 24782.223} C_VEL
LIN {X 0,Y 521.842,Z 612.619,A -85,B 0,C 180,E1 24779.181,E2 24779.181} C_VEL
LIN {X 0,Y 521.403,Z 654.512,A -85,B 0,C 180,E1 24778.542,E2 24778.542} C_VEL
LIN {X 0,Y 520.82,Z 675.959,A -85,B 0,C 180,E1 24778.013,E2 24778.013} C_VEL
LIN {X 0,Y 520.107,Z 696.653,A -85,B 0,C 180,E1 24777.289,E2 24777.289} C_VEL
LIN {X 0,Y 519.325,Z 714.871,A -85,B 0,C 180,E1 24776.458,E2 24776.458} C_VEL
LIN {X 0,Y 518.292,Z 733.832,A -85,B 0,C 180,E1 24775.357,E2 24775.357} C_VEL
LIN {X 0,Y 517.243,Z 751.976,A -85,B 0,C 180,E1 24774.071,E2 24774.071} C_VEL
LIN {X 0,Y 516.192,Z 769.069,A -85,B 0,C 180,E1 24772.622,E2 24772.622} C_VEL
LIN {X 0,Y 515.192,Z 785.082,A -85,B 0,C 180,E1 24771.013,E2 24771.013} C_VEL
LIN {X 0,Y 514.317,Z 799.521,A -85,B 0,C 180,E1 24769.298,E2 24769.298} C_VEL
LIN {X 0,Y 513.57,Z 812.811,A -85,B 0,C 180,E1 24767.446,E2 24767.446} C_VEL
LIN {X 0,Y 512.95,Z 825.379,A -85,B 0,C 180,E1 24765.372,E2 24765.372} C_VEL
LIN {X 0,Y 512.491,Z 836.334,A -85,B 0,C 180,E1 24763.195,E2 24763.195} C_VEL
LIN {X 0,Y 512.2,Z 845.252,A -85,B 0,C 180,E1 24761.029,E2 24761.029} C_VEL
LIN {X 0,Y 512.043,Z 852.402,A -85,B 0,C 180,E1 24758.865,E2 24758.865} C_VEL
LIN {X 0,Y 511.95,Z 858.005,A -85,B 0,C 180,E1 24756.617,E2 24756.617} C_VEL
LIN {X 0,Y 511.911,Z 861.928,A -85,B 0,C 180,E1 24754.369,E2 24754.369} C_VEL
LIN {X 0,Y 511.91,Z 864.305,A -85,B 0,C 180,E1 24752.015,E2 24752.015} C_VEL
LIN {X 0,Y 511.906,Z 864.962,A -85,B 0,C 180,E1 24749.776,E2 24749.776} C_VEL
LIN {X 0,Y 511.902,Z 864.032,A -85,B 0,C 180,E1 24747.537,E2 24747.537} C_VEL
LIN {X 0,Y 511.918,Z 861.448,A -85,B 0,C 180,E1 24745.295,E2 24745.295} C_VEL
LIN {X 0,Y 511.966,Z 857.245,A -85,B 0,C 180,E1 24743.045,E2 24743.045} C_VEL
LIN {X 0,Y 512.061,Z 851.327,A -85,B 0,C 180,E1 24740.787,E2 24740.787} C_VEL
LIN {X 0,Y 512.243,Z 844.012,A -85,B 0,C 180,E1 24738.63,E2 24738.63} C_VEL
LIN {X 0,Y 512.563,Z 834.785,A -85,B 0,C 180,E1 24736.463,E2 24736.463} C_VEL
LIN {X 0,Y 513.011,Z 824.109,A -85,B 0,C 180,E1 24734.398,E2 24734.398} C_VEL
LIN {X 0,Y 513.614,Z 812.042,A -85,B 0,C 180,E1 24732.438,E2 24732.438} C_VEL
LIN {X 0,Y 514.423,Z 797.669,A -85,B 0,C 180,E1 24730.47,E2 24730.47} C_VEL
LIN {X 0,Y 515.331,Z 782.612,A -85,B 0,C 180,E1 24728.727,E2 24728.727} C_VEL
LIN {X 0,Y 516.314,Z 767.011,A -85,B 0,C 180,E1 24727.189,E2 24727.189} C_VEL
LIN {X 0,Y 517.394,Z 749.769,A -85,B 0,C 180,E1 24725.755,E2 24725.755} C_VEL
LIN {X 0,Y 518.468,Z 731.124,A -85,B 0,C 180,E1 24724.469,E2 24724.469} C_VEL
LIN {X 0,Y 519.38,Z 713.518,A -85,B 0,C 180,E1 24723.474,E2 24723.474} C_VEL
LIN {X 0,Y 520.185,Z 694.39,A -85,B 0,C 180,E1 24722.625,E2 24722.625} C_VEL
LIN {X 0,Y 520.857,Z 674.152,A -85,B 0,C 180,E1 24721.935,E2 24721.935} C_VEL
LIN {X 0,Y 521.45,Z 652.683,A -85,B 0,C 180,E1 24721.42,E2 24721.42} C_VEL
LIN {X 0,Y 523.652,Z 413.389,A -85,B 0,C 180,E1 24717.89,E2 24717.89} C_VEL
LIN {X 0,Y 523.514,Z 402.54,A -85,B 0,C 180,E1 24717.711,E2 24717.711} C_VEL
LIN {X 0,Y 521.655,Z 388.415,A -85,B 0,C 180,E1 24717.348,E2 24717.348} C_VEL
LIN {X 0,Y 523.427,Z 334.157,A -85,B 0,C 180,E1 24713.961,E2 24713.961} C_VEL
LIN {X 0,Y 523.701,Z 325.929,A -85,B 0,C 180,E1 24713.44,E2 24713.44} C_VEL
LIN {X 0,Y 513.893,Z 302.019,A -85,B 0,C 180,E1 24711.101,E2 24711.101} C_VEL
LIN {X 0,Y 512.687,Z 298.891,A -85,B 0,C 180,E1 24710.736,E2 24710.736} C_VEL
LIN {X 0,Y 512.646,Z 298.619,A -85,B 0,C 180,E1 24709.008,E2 24709.008} C_VEL
LIN {X 0,Y 512.624,Z 298.616,A -85,B 0,C 180,E1 24705.551,E2 24705.551} C_VEL
LIN {X 0,Y 512.609,Z 298.606,A -85,B 0,C 180,E1 24702.143,E2 24702.143} C_VEL
LIN {X 0,Y 512.649,Z 298.631,A -85,B 0,C 180,E1 24698.728,E2 24698.728} C_VEL
LIN {X 0,Y 512.626,Z 298.607,A -85,B 0,C 180,E1 24695.263,E2 24695.263} C_VEL
LIN {X 0,Y 512.601,Z 298.628,A -85,B 0,C 180,E1 24691.911,E2 24691.911} C_VEL
LIN {X 0,Y 512.643,Z 298.629,A -85,B 0,C 180,E1 24688.545,E2 24688.545} C_VEL
LIN {X 0,Y 512.62,Z 298.629,A -85,B 0,C 180,E1 24685.163,E2 24685.163} C_VEL
LIN {X 0,Y 512.589,Z 298.63,A -85,B 0,C 180,E1 24681.753,E2 24681.753} C_VEL
LIN {X 0,Y 512.629,Z 298.623,A -85,B 0,C 180,E1 24678.419,E2 24678.419} C_VEL
LIN {X 0,Y 512.612,Z 298.63,A -85,B 0,C 180,E1 24675.035,E2 24675.035} C_VEL
LIN {X 0,Y 512.579,Z 298.631,A -85,B 0,C 180,E1 24671.704,E2 24671.704} C_VEL
LIN {X 0,Y 512.63,Z 298.621,A -85,B 0,C 180,E1 24668.411,E2 24668.411} C_VEL
LIN {X 0,Y 512.584,Z 298.632,A -85,B 0,C 180,E1 24665.148,E2 24665.148} C_VEL
LIN {X 0,Y 512.571,Z 298.629,A -85,B 0,C 180,E1 24661.676,E2 24661.676} C_VEL
LIN {X 0,Y 512.63,Z 298.625,A -85,B 0,C 180,E1 24658.435,E2 24658.435} C_VEL
LIN {X 0,Y 512.575,Z 298.631,A -85,B 0,C 180,E1 24655.076,E2 24655.076} C_VEL
LIN {X 0,Y 512.57,Z 298.621,A -85,B 0,C 180,E1 24651.587,E2 24651.587} C_VEL
LIN {X 0,Y 512.633,Z 298.63,A -85,B 0,C 180,E1 24648.263,E2 24648.263} C_VEL
LIN {X 0,Y 512.585,Z 298.623,A -85,B 0,C 180,E1 24644.963,E2 24644.963} C_VEL
LIN {X 0,Y 512.583,Z 298.627,A -85,B 0,C 180,E1 24641.438,E2 24641.438} C_VEL
LIN {X 0,Y 512.642,Z 298.63,A -85,B 0,C 180,E1 24638.128,E2 24638.128} C_VEL
LIN {X 0,Y 512.605,Z 298.622,A -85,B 0,C 180,E1 24634.712,E2 24634.712} C_VEL
LIN {X 0,Y 512.592,Z 298.627,A -85,B 0,C 180,E1 24631.324,E2 24631.324} C_VEL
LIN {X 0,Y 512.644,Z 298.627,A -85,B 0,C 180,E1 24627.96,E2 24627.96} C_VEL
LIN {X 0,Y 512.615,Z 298.63,A -85,B 0,C 180,E1 24624.598,E2 24624.598} C_VEL
LIN {X 0,Y 512.601,Z 298.628,A -85,B 0,C 180,E1 24621.235,E2 24621.235} C_VEL
LIN {X 0,Y 512.646,Z 298.628,A -85,B 0,C 180,E1 24617.827,E2 24617.827} C_VEL
LIN {X 0,Y 512.628,Z 298.61,A -85,B 0,C 180,E1 24614.443,E2 24614.443} C_VEL
LIN {X 0,Y 512.646,Z 298.604,A -85,B 0,C 180,E1 24614.05,E2 24614.05} C_VEL
LIN {X 0,Y 511.659,Z 298.729,A -85,B 0,C 180,E1 24613.189,E2 24613.189} C_VEL
LIN {X 0,Y 505.222,Z 299.555,A -85,B 0,C 180,E1 24610.77,E2 24610.77} C_VEL
LIN {X 0,Y 504.708,Z 299.611,A -85,B 0,C 180,E1 24610.139,E2 24610.139} C_VEL
LIN {X 0,Y 504.679,Z 299.619,A -85,B 0,C 180,E1 24606.642,E2 24606.642} C_VEL
LIN {X 0,Y 504.68,Z 299.612,A -85,B 0,C 180,E1 24603.066,E2 24603.066} C_VEL
LIN {X 0,Y 504.739,Z 299.824,A -85,B 0,C 180,E1 24601.797,E2 24601.797} C_VEL
LIN {X 0,Y 511.429,Z 319.703,A -85,B 0,C 180,E1 24599.085,E2 24599.085} C_VEL
LIN {X 0,Y 512.416,Z 323.723,A -85,B 0,C 180,E1 24598.589,E2 24598.589} C_VEL
LIN {X 0,Y 511.881,Z 338.043,A -85,B 0,C 180,E1 24597.206,E2 24597.206} C_VEL
LIN {X 0,Y 514.747,Z 351.959,A -85,B 0,C 180,E1 24596.804,E2 24596.804} C_VEL
LIN {X 0,Y 513.374,Z 549.16,A -85,B 0,C 180,E1 24594.017,E2 24594.017} C_VEL
LIN {X 0,Y 513.036,Z 567.95,A -85,B 0,C 180,E1 24593.533,E2 24593.533} C_VEL
LIN {X 0,Y 512.418,Z 586.083,A -85,B 0,C 180,E1 24592.848,E2 24592.848} C_VEL
LIN {X 0,Y 511.621,Z 603.28,A -85,B 0,C 180,E1 24591.977,E2 24591.977} C_VEL
LIN {X 0,Y 510.653,Z 619.451,A -85,B 0,C 180,E1 24590.937,E2 24590.937} C_VEL
LIN {X 0,Y 509.554,Z 635.433,A -85,B 0,C 180,E1 24589.659,E2 24589.659} C_VEL
LIN {X 0,Y 508.444,Z 650.127,A -85,B 0,C 180,E1 24588.22,E2 24588.22} C_VEL
LIN {X 0,Y 507.44,Z 662.883,A -85,B 0,C 180,E1 24586.718,E2 24586.718} C_VEL
LIN {X 0,Y 506.479,Z 675.107,A -85,B 0,C 180,E1 24584.987,E2 24584.987} C_VEL
LIN {X 0,Y 505.703,Z 685.853,A -85,B 0,C 180,E1 24583.142,E2 24583.142} C_VEL
LIN {X 0,Y 505.073,Z 695.186,A -85,B 0,C 180,E1 24581.186,E2 24581.186} C_VEL
LIN {X 0,Y 504.638,Z 703.041,A -85,B 0,C 180,E1 24579.12,E2 24579.12} C_VEL
LIN {X 0,Y 504.367,Z 709.364,A -85,B 0,C 180,E1 24576.945,E2 24576.945} C_VEL
LIN {X 0,Y 504.201,Z 714.057,A -85,B 0,C 180,E1 24574.663,E2 24574.663} C_VEL
LIN {X 0,Y 504.128,Z 716.767,A -85,B 0,C 180,E1 24572.501,E2 24572.501} C_VEL
LIN {X 0,Y 504.109,Z 717.852,A -85,B 0,C 180,E1 24570.341,E2 24570.341} C_VEL
LIN {X 0,Y 504.121,Z 717.337,A -85,B 0,C 180,E1 24568.182,E2 24568.182} C_VEL
LIN {X 0,Y 504.169,Z 715.167,A -85,B 0,C 180,E1 24565.984,E2 24565.984} C_VEL
LIN {X 0,Y 504.285,Z 711.422,A -85,B 0,C 180,E1 24563.854,E2 24563.854} C_VEL
LIN {X 0,Y 504.501,Z 706.194,A -85,B 0,C 180,E1 24561.796,E2 24561.796} C_VEL
LIN {X 0,Y 504.835,Z 699.254,A -85,B 0,C 180,E1 24559.732,E2 24559.732} C_VEL
LIN {X 0,Y 505.345,Z 690.915,A -85,B 0,C 180,E1 24557.778,E2 24557.778} C_VEL
LIN {X 0,Y 506.073,Z 680.59,A -85,B 0,C 180,E1 24555.819,E2 24555.819} C_VEL
LIN {X 0,Y 506.911,Z 669.493,A -85,B 0,C 180,E1 24554.088,E2 24554.088} C_VEL
LIN {X 0,Y 507.906,Z 657.034,A -85,B 0,C 180,E1 24552.471,E2 24552.471} C_VEL
LIN {X 0,Y 508.98,Z 643.116,A -85,B 0,C 180,E1 24550.969,E2 24550.969} C_VEL
LIN {X 0,Y 510.069,Z 628.183,A -85,B 0,C 180,E1 24549.639,E2 24549.639} C_VEL
LIN {X 0,Y 511.099,Z 612.257,A -85,B 0,C 180,E1 24548.482,E2 24548.482} C_VEL
LIN {X 0,Y 511.97,Z 596.327,A -85,B 0,C 180,E1 24547.555,E2 24547.555} C_VEL
LIN {X 0,Y 512.653,Z 579.704,A -85,B 0,C 180,E1 24546.799,E2 24546.799} C_VEL
LIN {X 0,Y 513.163,Z 561.572,A -85,B 0,C 180,E1 24546.192,E2 24546.192} C_VEL
LIN {X 0,Y 513.421,Z 543.114,A -85,B 0,C 180,E1 24545.788,E2 24545.788} C_VEL
LIN {X 0,Y 514.59,Z 350.216,A -85,B 0,C 180,E1 24543.068,E2 24543.068} C_VEL
LIN {X 0,Y 511.822,Z 337.494,A -85,B 0,C 180,E1 24542.673,E2 24542.673} C_VEL
LIN {X 0,Y 512.316,Z 322.47,A -85,B 0,C 180,E1 24541.181,E2 24541.181} C_VEL
LIN {X 0,Y 506.25,Z 304.508,A -85,B 0,C 180,E1 24538.781,E2 24538.781} C_VEL
LIN {X 0,Y 504.735,Z 299.815,A -85,B 0,C 180,E1 24538.102,E2 24538.102} C_VEL
LIN {X 0,Y 504.692,Z 299.608,A -85,B 0,C 180,E1 24534.657,E2 24534.657} C_VEL
LIN {X 0,Y 504.674,Z 299.6,A -85,B 0,C 180,E1 24531.096,E2 24531.096} C_VEL
LIN {X 0,Y 504.699,Z 299.606,A -85,B 0,C 180,E1 24527.642,E2 24527.642} C_VEL
LIN {X 0,Y 504.71,Z 299.609,A -85,B 0,C 180,E1 24524.056,E2 24524.056} C_VEL
LIN {X 0,Y 504.673,Z 299.616,A -85,B 0,C 180,E1 24520.643,E2 24520.643} C_VEL
LIN {X 0,Y 504.672,Z 299.619,A -85,B 0,C 180,E1 24517.177,E2 24517.177} C_VEL
LIN {X 0,Y 504.706,Z 299.611,A -85,B 0,C 180,E1 24513.693,E2 24513.693} C_VEL
LIN {X 0,Y 504.687,Z 299.615,A -85,B 0,C 180,E1 24510.213,E2 24510.213} C_VEL
LIN {X 0,Y 504.657,Z 299.619,A -85,B 0,C 180,E1 24506.855,E2 24506.855} C_VEL
LIN {X 0,Y 504.693,Z 299.616,A -85,B 0,C 180,E1 24503.466,E2 24503.466} C_VEL
LIN {X 0,Y 504.676,Z 299.614,A -85,B 0,C 180,E1 24500.106,E2 24500.106} C_VEL
LIN {X 0,Y 504.645,Z 299.62,A -85,B 0,C 180,E1 24496.696,E2 24496.696} C_VEL
LIN {X 0,Y 504.673,Z 299.616,A -85,B 0,C 180,E1 24493.287,E2 24493.287} C_VEL
LIN {X 0,Y 504.671,Z 299.619,A -85,B 0,C 180,E1 24489.926,E2 24489.926} C_VEL
LIN {X 0,Y 504.633,Z 299.621,A -85,B 0,C 180,E1 24486.599,E2 24486.599} C_VEL
LIN {X 0,Y 504.66,Z 299.61,A -85,B 0,C 180,E1 24483.18,E2 24483.18} C_VEL
LIN {X 0,Y 504.653,Z 299.622,A -85,B 0,C 180,E1 24479.887,E2 24479.887} C_VEL
LIN {X 0,Y 504.627,Z 299.615,A -85,B 0,C 180,E1 24476.479,E2 24476.479} C_VEL
LIN {X 0,Y 504.664,Z 299.613,A -85,B 0,C 180,E1 24473.059,E2 24473.059} C_VEL
LIN {X 0,Y 504.67,Z 299.619,A -85,B 0,C 180,E1 24469.729,E2 24469.729} C_VEL
LIN {X 0,Y 504.64,Z 299.609,A -85,B 0,C 180,E1 24466.363,E2 24466.363} C_VEL
LIN {X 0,Y 504.674,Z 299.615,A -85,B 0,C 180,E1 24462.95,E2 24462.95} C_VEL
LIN {X 0,Y 504.688,Z 299.619,A -85,B 0,C 180,E1 24459.562,E2 24459.562} C_VEL
LIN {X 0,Y 504.653,Z 299.615,A -85,B 0,C 180,E1 24456.16,E2 24456.16} C_VEL
LIN {X 0,Y 504.678,Z 299.612,A -85,B 0,C 180,E1 24452.764,E2 24452.764} C_VEL
LIN {X 0,Y 504.71,Z 299.611,A -85,B 0,C 180,E1 24449.289,E2 24449.289} C_VEL
LIN {X 0,Y 504.666,Z 299.618,A -85,B 0,C 180,E1 24445.897,E2 24445.897} C_VEL
LIN {X 0,Y 504.671,Z 299.613,A -85,B 0,C 180,E1 24442.395,E2 24442.395} C_VEL
LIN {X 0,Y 504.712,Z 299.592,A -85,B 0,C 180,E1 24439.004,E2 24439.004} C_VEL
LIN {X 0,Y 504.695,Z 299.618,A -85,B 0,C 180,E1 24435.468,E2 24435.468} C_VEL
LIN {X 0,Y 504.675,Z 299.621,A -85,B 0,C 180,E1 24432.017,E2 24432.017} C_VEL
LIN {X 0,Y 504.713,Z 299.862,A -85,B 0,C 180,E1 24429.836,E2 24429.836} C_VEL
LIN {X 0,Y 506.757,Z 305.082,A -85,B 0,C 180,E1 24429.248,E2 24429.248} C_VEL
LIN {X 0,Y 515.441,Z 326.149,A -85,B 0,C 180,E1 24427.131,E2 24427.131} C_VEL
LIN {X 0,Y 516.629,Z 329.342,A -85,B 0,C 180,E1 24426.831,E2 24426.831} C_VEL
LIN {X 0,Y 514.659,Z 383.058,A -85,B 0,C 180,E1 24423.419,E2 24423.419} C_VEL
LIN {X 0,Y 514.541,Z 389.313,A -85,B 0,C 180,E1 24423.054,E2 24423.054} C_VEL
LIN {X 0,Y 516.716,Z 406.891,A -85,B 0,C 180,E1 24422.635,E2 24422.635} C_VEL
LIN {X 0,Y 514.458,Z 621.066,A -85,B 0,C 180,E1 24419.42,E2 24419.42} C_VEL
LIN {X 0,Y 514.029,Z 654.431,A -85,B 0,C 180,E1 24418.889,E2 24418.889} C_VEL
LIN {X 0,Y 513.381,Z 675.365,A -85,B 0,C 180,E1 24418.36,E2 24418.36} C_VEL
LIN {X 0,Y 512.611,Z 695.931,A -85,B 0,C 180,E1 24417.628,E2 24417.628} C_VEL
LIN {X 0,Y 511.7,Z 715.853,A -85,B 0,C 180,E1 24416.705,E2 24416.705} C_VEL
LIN {X 0,Y 510.725,Z 734.559,A -85,B 0,C 180,E1 24415.635,E2 24415.635} C_VEL
LIN {X 0,Y 509.751,Z 752.602,A -85,B 0,C 180,E1 24414.386,E2 24414.386} C_VEL
LIN {X 0,Y 508.755,Z 767.669,A -85,B 0,C 180,E1 24413.109,E2 24413.109} C_VEL
LIN {X 0,Y 507.611,Z 784.278,A -85,B 0,C 180,E1 24411.431,E2 24411.431} C_VEL
LIN {X 0,Y 506.655,Z 798.595,A -85,B 0,C 180,E1 24409.722,E2 24409.722} C_VEL
LIN {X 0,Y 505.818,Z 812.04,A -85,B 0,C 180,E1 24407.841,E2 24407.841} C_VEL
LIN {X 0,Y 505.145,Z 824.107,A -85,B 0,C 180,E1 24405.851,E2 24405.851} C_VEL
LIN {X 0,Y 504.646,Z 834.787,A -85,B 0,C 180,E1 24403.754,E2 24403.754} C_VEL
LIN {X 0,Y 504.289,Z 844.009,A -85,B 0,C 180,E1 24401.551,E2 24401.551} C_VEL
LIN {X 0,Y 504.084,Z 851.323,A -85,B 0,C 180,E1 24399.36,E2 24399.36} C_VEL
LIN {X 0,Y 503.974,Z 857.243,A -85,B 0,C 180,E1 24397.065,E2 24397.065} C_VEL
LIN {X 0,Y 503.917,Z 861.608,A -85,B 0,C 180,E1 24394.666,E2 24394.666} C_VEL
LIN {X 0,Y 503.902,Z 864.101,A -85,B 0,C 180,E1 24392.388,E2 24392.388} C_VEL
LIN {X 0,Y 503.912,Z 864.984,A -85,B 0,C 180,E1 24390.114,E2 24390.114} C_VEL
LIN {X 0,Y 503.908,Z 864.236,A -85,B 0,C 180,E1 24387.839,E2 24387.839} C_VEL
LIN {X 0,Y 503.912,Z 861.926,A -85,B 0,C 180,E1 24385.562,E2 24385.562} C_VEL
LIN {X 0,Y 503.959,Z 858.006,A -85,B 0,C 180,E1 24383.278,E2 24383.278} C_VEL
LIN {X 0,Y 504.058,Z 852.379,A -85,B 0,C 180,E1 24380.985,E2 24380.985} C_VEL
LIN {X 0,Y 504.255,Z 844.847,A -85,B 0,C 180,E1 24378.68,E2 24378.68} C_VEL
LIN {X 0,Y 504.593,Z 835.819,A -85,B 0,C 180,E1 24376.478,E2 24376.478} C_VEL
LIN {X 0,Y 505.077,Z 825.378,A -85,B 0,C 180,E1 24374.382,E2 24374.382} C_VEL
LIN {X 0,Y 505.772,Z 812.811,A -85,B 0,C 180,E1 24372.276,E2 24372.276} C_VEL
LIN {X 0,Y 506.598,Z 799.52,A -85,B 0,C 180,E1 24370.396,E2 24370.396} C_VEL
LIN {X 0,Y 507.575,Z 784.829,A -85,B 0,C 180,E1 24368.628,E2 24368.628} C_VEL
LIN {X 0,Y 508.694,Z 768.567,A -85,B 0,C 180,E1 24366.975,E2 24366.975} C_VEL
LIN {X 0,Y 509.702,Z 753.356,A -85,B 0,C 180,E1 24365.674,E2 24365.674} C_VEL
LIN {X 0,Y 510.675,Z 735.504,A -85,B 0,C 180,E1 24364.424,E2 24364.424} C_VEL
LIN {X 0,Y 511.651,Z 717.032,A -85,B 0,C 180,E1 24363.354,E2 24363.354} C_VEL
LIN {X 0,Y 512.581,Z 696.692,A -85,B 0,C 180,E1 24362.402,E2 24362.402} C_VEL
LIN {X 0,Y 513.374,Z 675.607,A -85,B 0,C 180,E1 24361.648,E2 24361.648} C_VEL
LIN {X 0,Y 514.012,Z 654.92,A -85,B 0,C 180,E1 24361.122,E2 24361.122} C_VEL
LIN {X 0,Y 514.431,Z 623.804,A -85,B 0,C 180,E1 24360.62,E2 24360.62} C_VEL
LIN {X 0,Y 516.679,Z 409.85,A -85,B 0,C 180,E1 24357.41,E2 24357.41} C_VEL
LIN {X 0,Y 516.442,Z 403.292,A -85,B 0,C 180,E1 24357.29,E2 24357.29} C_VEL
LIN {X 0,Y 514.468,Z 387.957,A -85,B 0,C 180,E1 24356.891,E2 24356.891} C_VEL
LIN {X 0,Y 516.463,Z 333.855,A -85,B 0,C 180,E1 24353.459,E2 24353.459} C_VEL
LIN {X 0,Y 516.534,Z 328.811,A -85,B 0,C 180,E1 24353.126,E2 24353.126} C_VEL
LIN {X 0,Y 507.264,Z 306.162,A -85,B 0,C 180,E1 24350.87,E2 24350.87} C_VEL
LIN {X 0,Y 504.735,Z 299.994,A -85,B 0,C 180,E1 24350.189,E2 24350.189} C_VEL
LIN {X 0,Y 504.681,Z 299.598,A -85,B 0,C 180,E1 24349.707,E2 24349.707} C_VEL
LIN {X 0,Y 504.673,Z 299.599,A -85,B 0,C 180,E1 24346.15,E2 24346.15} C_VEL
LIN {X 0,Y 504.7,Z 299.596,A -85,B 0,C 180,E1 24342.651,E2 24342.651} C_VEL
LIN {X 0,Y 504.705,Z 299.616,A -85,B 0,C 180,E1 24339.195,E2 24339.195} C_VEL
LIN {X 0,Y 504.661,Z 299.594,A -85,B 0,C 180,E1 24335.765,E2 24335.765} C_VEL
LIN {X 0,Y 504.673,Z 299.618,A -85,B 0,C 180,E1 24332.226,E2 24332.226} C_VEL
LIN {X 0,Y 504.713,Z 299.62,A -85,B 0,C 180,E1 24328.776,E2 24328.776} C_VEL
LIN {X 0,Y 504.668,Z 299.619,A -85,B 0,C 180,E1 24325.337,E2 24325.337} C_VEL
LIN {X 0,Y 504.653,Z 299.62,A -85,B 0,C 180,E1 24321.868,E2 24321.868} C_VEL
LIN {X 0,Y 504.695,Z 299.611,A -85,B 0,C 180,E1 24318.48,E2 24318.48} C_VEL
LIN {X 0,Y 504.673,Z 299.619,A -85,B 0,C 180,E1 24315.042,E2 24315.042} C_VEL
LIN {X 0,Y 504.64,Z 299.62,A -85,B 0,C 180,E1 24311.659,E2 24311.659} C_VEL
LIN {X 0,Y 504.679,Z 299.61,A -85,B 0,C 180,E1 24308.315,E2 24308.315} C_VEL
LIN {X 0,Y 504.656,Z 299.621,A -85,B 0,C 180,E1 24305.001,E2 24305.001} C_VEL
LIN {X 0,Y 504.63,Z 299.618,A -85,B 0,C 180,E1 24301.589,E2 24301.589} C_VEL
LIN {X 0,Y 504.678,Z 299.613,A -85,B 0,C 180,E1 24298.297,E2 24298.297} C_VEL
LIN {X 0,Y 504.65,Z 299.62,A -85,B 0,C 180,E1 24294.885,E2 24294.885} C_VEL
LIN {X 0,Y 504.629,Z 299.609,A -85,B 0,C 180,E1 24291.454,E2 24291.454} C_VEL
LIN {X 0,Y 504.676,Z 299.619,A -85,B 0,C 180,E1 24288.109,E2 24288.109} C_VEL
LIN {X 0,Y 504.66,Z 299.612,A -85,B 0,C 180,E1 24284.762,E2 24284.762} C_VEL
LIN {X 0,Y 504.643,Z 299.616,A -85,B 0,C 180,E1 24281.398,E2 24281.398} C_VEL
LIN {X 0,Y 504.689,Z 299.618,A -85,B 0,C 180,E1 24277.994,E2 24277.994} C_VEL
LIN {X 0,Y 504.675,Z 299.61,A -85,B 0,C 180,E1 24274.608,E2 24274.608} C_VEL
LIN {X 0,Y 504.652,Z 299.616,A -85,B 0,C 180,E1 24271.219,E2 24271.219} C_VEL
LIN {X 0,Y 504.702,Z 299.616,A -85,B 0,C 180,E1 24267.931,E2 24267.931} C_VEL
LIN {X 0,Y 504.684,Z 299.619,A -85,B 0,C 180,E1 24264.512,E2 24264.512} C_VEL
LIN {X 0,Y 504.66,Z 299.618,A -85,B 0,C 180,E1 24261.093,E2 24261.093} C_VEL
LIN {X 0,Y 504.693,Z 299.617,A -85,B 0,C 180,E1 24257.641,E2 24257.641} C_VEL
LIN {X 0,Y 504.704,Z 299.592,A -85,B 0,C 180,E1 24254.18,E2 24254.18} C_VEL
LIN {X 0,Y 504.676,Z 299.623,A -85,B 0,C 180,E1 24250.677,E2 24250.677} C_VEL
LIN {X 0,Y 504.708,Z 299.611,A -85,B 0,C 180,E1 24250.139,E2 24250.139} C_VEL
LIN {X 0,Y 503.738,Z 299.726,A -85,B 0,C 180,E1 24249.265,E2 24249.265} C_VEL
LIN {X 0,Y 497.288,Z 300.549,A -85,B 0,C 180,E1 24246.807,E2 24246.807} C_VEL
LIN {X 0,Y 496.766,Z 300.607,A -85,B 0,C 180,E1 24246.166,E2 24246.166} C_VEL
LIN {X 0,Y 496.742,Z 300.61,A -85,B 0,C 180,E1 24242.644,E2 24242.644} C_VEL
LIN {X 0,Y 496.803,Z 300.914,A -85,B 0,C 180,E1 24242.336,E2 24242.336} C_VEL
LIN {X 0,Y 503.421,Z 320.289,A -85,B 0,C 180,E1 24239.639,E2 24239.639} C_VEL
LIN {X 0,Y 505.217,Z 326.167,A -85,B 0,C 180,E1 24238.874,E2 24238.874} C_VEL
LIN {X 0,Y 504.756,Z 338.534,A -85,B 0,C 180,E1 24237.677,E2 24237.677} C_VEL
LIN {X 0,Y 507.823,Z 353.46,A -85,B 0,C 180,E1 24237.237,E2 24237.237} C_VEL
LIN {X 0,Y 506.34,Z 550.11,A -85,B 0,C 180,E1 24234.433,E2 24234.433} C_VEL
LIN {X 0,Y 505.988,Z 568.991,A -85,B 0,C 180,E1 24233.943,E2 24233.943} C_VEL
LIN {X 0,Y 505.342,Z 587.22,A -85,B 0,C 180,E1 24233.248,E2 24233.248} C_VEL
LIN {X 0,Y 504.503,Z 604.507,A -85,B 0,C 180,E1 24232.365,E2 24232.365} C_VEL
LIN {X 0,Y 503.482,Z 620.785,A -85,B 0,C 180,E1 24231.31,E2 24231.31} C_VEL
LIN {X 0,Y 502.336,Z 636.582,A -85,B 0,C 180,E1 24230.035,E2 24230.035} C_VEL
LIN {X 0,Y 501.163,Z 650.98,A -85,B 0,C 180,E1 24228.615,E2 24228.615} C_VEL
LIN {X 0,Y 500.057,Z 663.784,A -85,B 0,C 180,E1 24227.093,E2 24227.093} C_VEL
LIN {X 0,Y 498.982,Z 676.037,A -85,B 0,C 180,E1 24225.337,E2 24225.337} C_VEL
LIN {X 0,Y 498.102,Z 686.807,A -85,B 0,C 180,E1 24223.465,E2 24223.465} C_VEL
LIN {X 0,Y 497.375,Z 696.144,A -85,B 0,C 180,E1 24221.479,E2 24221.479} C_VEL
LIN {X 0,Y 496.862,Z 704.015,A -85,B 0,C 180,E1 24219.381,E2 24219.381} C_VEL
LIN {X 0,Y 496.546,Z 710.089,A -85,B 0,C 180,E1 24217.288,E2 24217.288} C_VEL
LIN {X 0,Y 496.333,Z 714.727,A -85,B 0,C 180,E1 24215.085,E2 24215.085} C_VEL
LIN {X 0,Y 496.233,Z 717.667,A -85,B 0,C 180,E1 24212.887,E2 24212.887} C_VEL
LIN {X 0,Y 496.205,Z 718.991,A -85,B 0,C 180,E1 24210.693,E2 24210.693} C_VEL
LIN {X 0,Y 496.209,Z 718.732,A -85,B 0,C 180,E1 24208.499,E2 24208.499} C_VEL
LIN {X 0,Y 496.259,Z 716.885,A -85,B 0,C 180,E1 24206.304,E2 24206.304} C_VEL
LIN {X 0,Y 496.39,Z 713.394,A -85,B 0,C 180,E1 24204.104,E2 24204.104} C_VEL
LIN {X 0,Y 496.644,Z 708.164,A -85,B 0,C 180,E1 24201.899,E2 24201.899} C_VEL
LIN {X 0,Y 497.035,Z 701.064,A -85,B 0,C 180,E1 24199.687,E2 24199.687} C_VEL
LIN {X 0,Y 497.603,Z 692.919,A -85,B 0,C 180,E1 24197.703,E2 24197.703} C_VEL
LIN {X 0,Y 498.407,Z 682.823,A -85,B 0,C 180,E1 24195.715,E2 24195.715} C_VEL
LIN {X 0,Y 499.319,Z 671.974,A -85,B 0,C 180,E1 24193.959,E2 24193.959} C_VEL
LIN {X 0,Y 500.393,Z 659.804,A -85,B 0,C 180,E1 24192.32,E2 24192.32} C_VEL
LIN {X 0,Y 501.545,Z 646.213,A -85,B 0,C 180,E1 24190.796,E2 24190.796} C_VEL
LIN {X 0,Y 502.752,Z 630.927,A -85,B 0,C 180,E1 24189.39,E2 24189.39} C_VEL
LIN {X 0,Y 503.84,Z 615.244,A -85,B 0,C 180,E1 24188.217,E2 24188.217} C_VEL
LIN {X 0,Y 504.815,Z 598.584,A -85,B 0,C 180,E1 24187.219,E2 24187.219} C_VEL
LIN {X 0,Y 505.561,Z 581.515,A -85,B 0,C 180,E1 24186.423,E2 24186.423} C_VEL
LIN {X 0,Y 506.118,Z 562.925,A -85,B 0,C 180,E1 24185.789,E2 24185.789} C_VEL
LIN {X 0,Y 506.384,Z 544.23,A -85,B 0,C 180,E1 24185.374,E2 24185.374} C_VEL
LIN {X 0,Y 507.687,Z 351.726,A -85,B 0,C 180,E1 24182.635,E2 24182.635} C_VEL
LIN {X 0,Y 504.693,Z 337.826,A -85,B 0,C 180,E1 24182.19,E2 24182.19} C_VEL
LIN {X 0,Y 505.226,Z 325.83,A -85,B 0,C 180,E1 24180.997,E2 24180.997} C_VEL
LIN {X 0,Y 498.839,Z 306.698,A -85,B 0,C 180,E1 24178.415,E2 24178.415} C_VEL
LIN {X 0,Y 496.779,Z 300.776,A -85,B 0,C 180,E1 24177.529,E2 24177.529} C_VEL
LIN {X 0,Y 496.768,Z 300.601,A -85,B 0,C 180,E1 24174.149,E2 24174.149} C_VEL
LIN {X 0,Y 496.748,Z 300.59,A -85,B 0,C 180,E1 24170.617,E2 24170.617} C_VEL
LIN {X 0,Y 496.735,Z 300.589,A -85,B 0,C 180,E1 24167.112,E2 24167.112} C_VEL
LIN {X 0,Y 496.76,Z 300.607,A -85,B 0,C 180,E1 24163.567,E2 24163.567} C_VEL
LIN {X 0,Y 496.771,Z 300.603,A -85,B 0,C 180,E1 24160.096,E2 24160.096} C_VEL
LIN {X 0,Y 496.728,Z 300.606,A -85,B 0,C 180,E1 24156.715,E2 24156.715} C_VEL
LIN {X 0,Y 496.728,Z 300.608,A -85,B 0,C 180,E1 24153.14,E2 24153.14} C_VEL
LIN {X 0,Y 496.772,Z 300.598,A -85,B 0,C 180,E1 24149.678,E2 24149.678} C_VEL
LIN {X 0,Y 496.744,Z 300.606,A -85,B 0,C 180,E1 24146.156,E2 24146.156} C_VEL
LIN {X 0,Y 496.712,Z 300.609,A -85,B 0,C 180,E1 24142.736,E2 24142.736} C_VEL
LIN {X 0,Y 496.73,Z 300.601,A -85,B 0,C 180,E1 24139.263,E2 24139.263} C_VEL
LIN {X 0,Y 496.756,Z 300.607,A -85,B 0,C 180,E1 24135.829,E2 24135.829} C_VEL
LIN {X 0,Y 496.702,Z 300.607,A -85,B 0,C 180,E1 24132.439,E2 24132.439} C_VEL
LIN {X 0,Y 496.704,Z 300.597,A -85,B 0,C 180,E1 24128.917,E2 24128.917} C_VEL
LIN {X 0,Y 496.757,Z 300.61,A -85,B 0,C 180,E1 24125.544,E2 24125.544} C_VEL
LIN {X 0,Y 496.703,Z 300.6,A -85,B 0,C 180,E1 24122.077,E2 24122.077} C_VEL
LIN {X 0,Y 496.688,Z 300.606,A -85,B 0,C 180,E1 24118.616,E2 24118.616} C_VEL
LIN {X 0,Y 496.73,Z 300.61,A -85,B 0,C 180,E1 24115.151,E2 24115.151} C_VEL
LIN {X 0,Y 496.724,Z 300.6,A -85,B 0,C 180,E1 24111.784,E2 24111.784} C_VEL
LIN {X 0,Y 496.7,Z 300.61,A -85,B 0,C 180,E1 24108.387,E2 24108.387} C_VEL
LIN {X 0,Y 496.731,Z 300.609,A -85,B 0,C 180,E1 24104.95,E2 24104.95} C_VEL
LIN {X 0,Y 496.746,Z 300.6,A -85,B 0,C 180,E1 24101.578,E2 24101.578} C_VEL
LIN {X 0,Y 496.714,Z 300.608,A -85,B 0,C 180,E1 24098.116,E2 24098.116} C_VEL
LIN {X 0,Y 496.725,Z 300.608,A -85,B 0,C 180,E1 24094.612,E2 24094.612} C_VEL
LIN {X 0,Y 496.772,Z 300.607,A -85,B 0,C 180,E1 24091.115,E2 24091.115} C_VEL
LIN {X 0,Y 496.742,Z 300.608,A -85,B 0,C 180,E1 24087.628,E2 24087.628} C_VEL
LIN {X 0,Y 496.721,Z 300.58,A -85,B 0,C 180,E1 24084.144,E2 24084.144} C_VEL
LIN {X 0,Y 496.753,Z 300.605,A -85,B 0,C 180,E1 24080.652,E2 24080.652} C_VEL
LIN {X 0,Y 496.77,Z 300.588,A -85,B 0,C 180,E1 24077.105,E2 24077.105} C_VEL
LIN {X 0,Y 496.747,Z 300.584,A -85,B 0,C 180,E1 24073.564,E2 24073.564} C_VEL
LIN {X 0,Y 496.783,Z 300.823,A -85,B 0,C 180,E1 24070.433,E2 24070.433} C_VEL
LIN {X 0,Y 498.108,Z 304.176,A -85,B 0,C 180,E1 24070.023,E2 24070.023} C_VEL
LIN {X 0,Y 507.808,Z 327.665,A -85,B 0,C 180,E1 24067.589,E2 24067.589} C_VEL
LIN {X 0,Y 509.568,Z 332.753,A -85,B 0,C 180,E1 24067.11,E2 24067.11} C_VEL
LIN {X 0,Y 507.393,Z 385.651,A -85,B 0,C 180,E1 24063.697,E2 24063.697} C_VEL
LIN {X 0,Y 507.432,Z 389.258,A -85,B 0,C 180,E1 24063.512,E2 24063.512} C_VEL
LIN {X 0,Y 509.721,Z 408.002,A -85,B 0,C 180,E1 24063.057,E2 24063.057} C_VEL
LIN {X 0,Y 507.125,Z 625.41,A -85,B 0,C 180,E1 24059.728,E2 24059.728} C_VEL
LIN {X 0,Y 506.653,Z 654.921,A -85,B 0,C 180,E1 24059.232,E2 24059.232} C_VEL
LIN {X 0,Y 505.933,Z 675.538,A -85,B 0,C 180,E1 24058.691,E2 24058.691} C_VEL
LIN {X 0,Y 505.099,Z 695.941,A -85,B 0,C 180,E1 24057.946,E2 24057.946} C_VEL
LIN {X 0,Y 504.034,Z 717.336,A -85,B 0,C 180,E1 24056.924,E2 24056.924} C_VEL
LIN {X 0,Y 502.863,Z 737.943,A -85,B 0,C 180,E1 24055.686,E2 24055.686} C_VEL
LIN {X 0,Y 501.734,Z 756.879,A -85,B 0,C 180,E1 24054.296,E2 24054.296} C_VEL
LIN {X 0,Y 500.647,Z 774.041,A -85,B 0,C 180,E1 24052.795,E2 24052.795} C_VEL
LIN {X 0,Y 499.69,Z 788.423,A -85,B 0,C 180,E1 24051.295,E2 24051.295} C_VEL
LIN {X 0,Y 498.704,Z 802.24,A -85,B 0,C 180,E1 24049.558,E2 24049.558} C_VEL
LIN {X 0,Y 497.792,Z 815.873,A -85,B 0,C 180,E1 24047.534,E2 24047.534} C_VEL
LIN {X 0,Y 497.08,Z 827.917,A -85,B 0,C 180,E1 24045.397,E2 24045.397} C_VEL
LIN {X 0,Y 496.574,Z 837.876,A -85,B 0,C 180,E1 24043.27,E2 24043.27} C_VEL
LIN {X 0,Y 496.237,Z 846.465,A -85,B 0,C 180,E1 24041.035,E2 24041.035} C_VEL
LIN {X 0,Y 496.043,Z 853.594,A -85,B 0,C 180,E1 24038.695,E2 24038.695} C_VEL
LIN {X 0,Y 495.949,Z 858.727,A -85,B 0,C 180,E1 24036.482,E2 24036.482} C_VEL
LIN {X 0,Y 495.915,Z 862.405,A -85,B 0,C 180,E1 24034.162,E2 24034.162} C_VEL
LIN {X 0,Y 495.908,Z 864.44,A -85,B 0,C 180,E1 24031.849,E2 24031.849} C_VEL
LIN {X 0,Y 495.901,Z 864.894,A -85,B 0,C 180,E1 24029.422,E2 24029.422} C_VEL
LIN {X 0,Y 495.915,Z 863.732,A -85,B 0,C 180,E1 24027.111,E2 24027.111} C_VEL
LIN {X 0,Y 495.931,Z 860.968,A -85,B 0,C 180,E1 24024.795,E2 24024.795} C_VEL
LIN {X 0,Y 495.989,Z 856.482,A -85,B 0,C 180,E1 24022.471,E2 24022.471} C_VEL
LIN {X 0,Y 496.124,Z 850.267,A -85,B 0,C 180,E1 24020.137,E2 24020.137} C_VEL
LIN {X 0,Y 496.391,Z 842.176,A -85,B 0,C 180,E1 24017.79,E2 24017.79} C_VEL
LIN {X 0,Y 496.806,Z 833.135,A -85,B 0,C 180,E1 24015.668,E2 24015.668} C_VEL
LIN {X 0,Y 497.423,Z 821.957,A -85,B 0,C 180,E1 24013.497,E2 24013.497} C_VEL
LIN {X 0,Y 498.244,Z 808.955,A -85,B 0,C 180,E1 24011.394,E2 24011.394} C_VEL
LIN {X 0,Y 499.224,Z 794.89,A -85,B 0,C 180,E1 24009.483,E2 24009.483} C_VEL
LIN {X 0,Y 500.184,Z 781.316,A -85,B 0,C 180,E1 24007.926,E2 24007.926} C_VEL
LIN {X 0,Y 501.2,Z 765.293,A -85,B 0,C 180,E1 24006.409,E2 24006.409} C_VEL
LIN {X 0,Y 502.312,Z 747.42,A -85,B 0,C 180,E1 24004.978,E2 24004.978} C_VEL
LIN {X 0,Y 503.421,Z 728.435,A -85,B 0,C 180,E1 24003.711,E2 24003.711} C_VEL
LIN {X 0,Y 504.487,Z 708.483,A -85,B 0,C 180,E1 24002.626,E2 24002.626} C_VEL
LIN {X 0,Y 505.373,Z 689.011,A -85,B 0,C 180,E1 24001.781,E2 24001.781} C_VEL
LIN {X 0,Y 506.229,Z 667.949,A -85,B 0,C 180,E1 24001.089,E2 24001.089} C_VEL
LIN {X 0,Y 506.843,Z 646.696,A -85,B 0,C 180,E1 24000.605,E2 24000.605} C_VEL
LIN {X 0,Y 509.576,Z 418.361,A -85,B 0,C 180,E1 23997.104,E2 23997.104} C_VEL
LIN {X 0,Y 509.53,Z 404.975,A -85,B 0,C 180,E1 23996.881,E2 23996.881} C_VEL
LIN {X 0,Y 507.314,Z 387.543,A -85,B 0,C 180,E1 23996.424,E2 23996.424} C_VEL
LIN {X 0,Y 509.493,Z 334.564,A -85,B 0,C 180,E1 23993.008,E2 23993.008} C_VEL
LIN {X 0,Y 509.381,Z 331.679,A -85,B 0,C 180,E1 23992.803,E2 23992.803} C_VEL
LIN {X 0,Y 500.614,Z 310.145,A -85,B 0,C 180,E1 23990.618,E2 23990.618} C_VEL
LIN {X 0,Y 496.816,Z 301.036,A -85,B 0,C 180,E1 23989.608,E2 23989.608} C_VEL
LIN {X 0,Y 496.77,Z 300.586,A -85,B 0,C 180,E1 23989.3,E2 23989.3} C_VEL
LIN {X 0,Y 496.735,Z 300.588,A -85,B 0,C 180,E1 23985.772,E2 23985.772} C_VEL
LIN {X 0,Y 496.733,Z 300.581,A -85,B 0,C 180,E1 23982.208,E2 23982.208} C_VEL
LIN {X 0,Y 496.772,Z 300.608,A -85,B 0,C 180,E1 23978.752,E2 23978.752} C_VEL
LIN {X 0,Y 496.754,Z 300.582,A -85,B 0,C 180,E1 23975.198,E2 23975.198} C_VEL
LIN {X 0,Y 496.722,Z 300.605,A -85,B 0,C 180,E1 23971.829,E2 23971.829} C_VEL
LIN {X 0,Y 496.746,Z 300.605,A -85,B 0,C 180,E1 23968.361,E2 23968.361} C_VEL
LIN {X 0,Y 496.771,Z 300.608,A -85,B 0,C 180,E1 23964.809,E2 23964.809} C_VEL
LIN {X 0,Y 496.721,Z 300.607,A -85,B 0,C 180,E1 23961.367,E2 23961.367} C_VEL
LIN {X 0,Y 496.71,Z 300.605,A -85,B 0,C 180,E1 23957.805,E2 23957.805} C_VEL
LIN {X 0,Y 496.754,Z 300.599,A -85,B 0,C 180,E1 23954.453,E2 23954.453} C_VEL
LIN {X 0,Y 496.727,Z 300.608,A -85,B 0,C 180,E1 23951.024,E2 23951.024} C_VEL
LIN {X 0,Y 496.697,Z 300.603,A -85,B 0,C 180,E1 23947.635,E2 23947.635} C_VEL
LIN {X 0,Y 496.735,Z 300.604,A -85,B 0,C 180,E1 23944.271,E2 23944.271} C_VEL
LIN {X 0,Y 496.727,Z 300.606,A -85,B 0,C 180,E1 23940.807,E2 23940.807} C_VEL
LIN {X 0,Y 496.686,Z 300.601,A -85,B 0,C 180,E1 23937.461,E2 23937.461} C_VEL
LIN {X 0,Y 496.715,Z 300.61,A -85,B 0,C 180,E1 23933.991,E2 23933.991} C_VEL
LIN {X 0,Y 496.723,Z 300.597,A -85,B 0,C 180,E1 23930.733,E2 23930.733} C_VEL
LIN {X 0,Y 496.695,Z 300.609,A -85,B 0,C 180,E1 23927.325,E2 23927.325} C_VEL
LIN {X 0,Y 496.725,Z 300.609,A -85,B 0,C 180,E1 23923.872,E2 23923.872} C_VEL
LIN {X 0,Y 496.759,Z 300.597,A -85,B 0,C 180,E1 23920.381,E2 23920.381} C_VEL
LIN {X 0,Y 496.712,Z 300.61,A -85,B 0,C 180,E1 23917.013,E2 23917.013} C_VEL
LIN {X 0,Y 496.718,Z 300.608,A -85,B 0,C 180,E1 23913.457,E2 23913.457} C_VEL
LIN {X 0,Y 496.775,Z 300.599,A -85,B 0,C 180,E1 23910.056,E2 23910.056} C_VEL
LIN {X 0,Y 496.745,Z 300.604,A -85,B 0,C 180,E1 23906.529,E2 23906.529} C_VEL
LIN {X 0,Y 496.723,Z 300.608,A -85,B 0,C 180,E1 23903.044,E2 23903.044} C_VEL
LIN {X 0,Y 496.742,Z 300.605,A -85,B 0,C 180,E1 23899.537,E2 23899.537} C_VEL
LIN {X 0,Y 496.771,Z 300.6,A -85,B 0,C 180,E1 23896.021,E2 23896.021} C_VEL
LIN {X 0,Y 496.742,Z 300.592,A -85,B 0,C 180,E1 23892.549,E2 23892.549} C_VEL
LIN {X 0,Y 496.731,Z 300.589,A -85,B 0,C 180,E1 23889.015,E2 23889.015} C_VEL
LIN {X 0,Y 496.766,Z 300.607,A -85,B 0,C 180,E1 23886.166,E2 23886.166} C_VEL
LIN {X 0,Y 495.775,Z 300.723,A -85,B 0,C 180,E1 23885.575,E2 23885.575} C_VEL
LIN {X 0,Y 489.373,Z 301.503,A -85,B 0,C 180,E1 23883.971,E2 23883.971} C_VEL
LIN {X 0,Y 488.825,Z 301.575,A -85,B 0,C 180,E1 23883.535,E2 23883.535} C_VEL
LIN {X 0,Y 488.844,Z 301.894,A -85,B 0,C 180,E1 23882.925,E2 23882.925} C_VEL
LIN {X 0,Y 495.742,Z 321.797,A -85,B 0,C 180,E1 23880.088,E2 23880.088} C_VEL
LIN {X 0,Y 498.02,Z 328.793,A -85,B 0,C 180,E1 23879.151,E2 23879.151} C_VEL
LIN {X 0,Y 497.67,Z 339.087,A -85,B 0,C 180,E1 23878.159,E2 23878.159} C_VEL
LIN {X 0,Y 500.93,Z 354.775,A -85,B 0,C 180,E1 23877.684,E2 23877.684} C_VEL
LIN {X 0,Y 499.307,Z 551.109,A -85,B 0,C 180,E1 23874.855,E2 23874.855} C_VEL
LIN {X 0,Y 498.934,Z 570.008,A -85,B 0,C 180,E1 23874.358,E2 23874.358} C_VEL
LIN {X 0,Y 498.261,Z 588.121,A -85,B 0,C 180,E1 23873.661,E2 23873.661} C_VEL
LIN {X 0,Y 497.371,Z 605.484,A -85,B 0,C 180,E1 23872.766,E2 23872.766} C_VEL
LIN {X 0,Y 496.289,Z 621.829,A -85,B 0,C 180,E1 23871.696,E2 23871.696} C_VEL
LIN {X 0,Y 495.057,Z 637.793,A -85,B 0,C 180,E1 23870.395,E2 23870.395} C_VEL
LIN {X 0,Y 493.846,Z 651.827,A -85,B 0,C 180,E1 23869.001,E2 23869.001} C_VEL
LIN {X 0,Y 492.585,Z 665.464,A -85,B 0,C 180,E1 23867.36,E2 23867.36} C_VEL
LIN {X 0,Y 491.425,Z 677.665,A -85,B 0,C 180,E1 23865.579,E2 23865.579} C_VEL
LIN {X 0,Y 490.457,Z 688.347,A -85,B 0,C 180,E1 23863.679,E2 23863.679} C_VEL
LIN {X 0,Y 489.651,Z 697.598,A -85,B 0,C 180,E1 23861.663,E2 23861.663} C_VEL
LIN {X 0,Y 489.071,Z 705.39,A -85,B 0,C 180,E1 23859.532,E2 23859.532} C_VEL
LIN {X 0,Y 488.685,Z 711.677,A -85,B 0,C 180,E1 23857.288,E2 23857.288} C_VEL
LIN {X 0,Y 488.438,Z 716.36,A -85,B 0,C 180,E1 23854.932,E2 23854.932} C_VEL
LIN {X 0,Y 488.324,Z 719.198,A -85,B 0,C 180,E1 23852.582,E2 23852.582} C_VEL
LIN {X 0,Y 488.291,Z 720.256,A -85,B 0,C 180,E1 23850.352,E2 23850.352} C_VEL
LIN {X 0,Y 488.309,Z 719.751,A -85,B 0,C 180,E1 23848.123,E2 23848.123} C_VEL
LIN {X 0,Y 488.383,Z 717.672,A -85,B 0,C 180,E1 23845.891,E2 23845.891} C_VEL
LIN {X 0,Y 488.554,Z 713.959,A -85,B 0,C 180,E1 23843.655,E2 23843.655} C_VEL
LIN {X 0,Y 488.876,Z 708.516,A -85,B 0,C 180,E1 23841.414,E2 23841.414} C_VEL
LIN {X 0,Y 489.338,Z 701.622,A -85,B 0,C 180,E1 23839.284,E2 23839.284} C_VEL
LIN {X 0,Y 490.019,Z 693.261,A -85,B 0,C 180,E1 23837.25,E2 23837.25} C_VEL
LIN {X 0,Y 490.925,Z 683.109,A -85,B 0,C 180,E1 23835.251,E2 23835.251} C_VEL
LIN {X 0,Y 491.955,Z 672.054,A -85,B 0,C 180,E1 23833.469,E2 23833.469} C_VEL
LIN {X 0,Y 493.138,Z 659.594,A -85,B 0,C 180,E1 23831.806,E2 23831.806} C_VEL
LIN {X 0,Y 494.334,Z 646.199,A -85,B 0,C 180,E1 23830.32,E2 23830.32} C_VEL
LIN {X 0,Y 495.572,Z 631.291,A -85,B 0,C 180,E1 23828.954,E2 23828.954} C_VEL
LIN {X 0,Y 496.73,Z 615.382,A -85,B 0,C 180,E1 23827.765,E2 23827.765} C_VEL
